		VIS.sBadPackageReason1 :=	CONCAT(CONCAT(CONCAT(CONCAT(CONCAT(CONCAT(sBadPackage1Reason1,':'),INT_TO_STRING(iBadPackage1ReasonCount1)),';'),sBadPackage2Reason1),':'),INT_TO_STRING(iBadPackage2ReasonCount1));
		VIS.sBadPackageReason2 :=	CONCAT(CONCAT(CONCAT(CONCAT(CONCAT(CONCAT(sBadPackage1Reason2,':'),INT_TO_STRING(iBadPackage1ReasonCount2)),';'),sBadPackage2Reason2),':'),INT_TO_STRING(iBadPackage2ReasonCount2));
		VIS.sBadPackageReason3 :=	CONCAT(CONCAT(CONCAT(CONCAT(CONCAT(CONCAT(sBadPackage1Reason3,':'),INT_TO_STRING(iBadPackage1ReasonCount3)),';'),sBadPackage2Reason3),':'),INT_TO_STRING(iBadPackage2ReasonCount3));
		
		
		bAddBadPackageReason	:= FALSE;
		
*)
END_ACTION

ACTION aCycleLogicHMI:
(*
Nazwa:			aCycleLogicHMI
Opis:			Wypracowanie sygnałów dla HMI
Wersja:			v0.2
Data:			2019-07-16
Autor:			DP
Urzadzenia:		
Konfiguracja:	
Info:
-daodano wbijak nasadek
*)



(*Dane do wykresów*)
//Wykresy wag i ilości wydozowanych
VIS.lrDispencer1DoseVolumeCV;			//Wartość wydana dozownika 1
VIS.lrDispencer2DoseVolumeCV;			//Wartość wydana dozownika 2
VIS.lrDispencer3DoseVolumeCV;			//Wartość wydana dozownika 3
VIS.lrDispencer4DoseVolumeCV;			//Wartość wydana dozownika 4
VIS.lrDispencer1WeightMeasured;			//Wartoć zmierzonej wagi dozowika 1 	
VIS.lrDispencer2WeightMeasured;			//Wartoć zmierzonej wagi dozowika 2	
VIS.lrDispencer3WeightMeasured;			//Wartoć zmierzonej wagi dozowika 3	
VIS.lrDispencer4WeightMeasured;			//Wartoć zmierzonej wagi dozowika 4	


//Pomiary przebiegu dozowania dozownika 1
VIS.bHMIDispencer1SuckingValveActuator					:= P02_Dispencers.QbDispencer1SuckingValveActuator;
VIS.bHMIDispencer1DosingValveActuator					:= P02_Dispencers.QbDispencer1DosingValveActuator;
VIS.bHMIDispencer1DropCatcherValveActuator				:= P02_Dispencers.QbDispencer1DropCatcherValveActuator;

//Pomiary przebiegu dozowania dozownika 2
VIS.bHMIDispencer2SuckingValveActuator					:= P02_Dispencers.QbDispencer2SuckingValveActuator;
VIS.bHMIDispencer2DosingValveActuator					:= P02_Dispencers.QbDispencer2DosingValveActuator;
VIS.bHMIDispencer2DropCatcherValveActuator				:= P02_Dispencers.QbDispencer2DropCatcherValveActuator;

//Pomiary przebiegu dozowania dozownika 3
VIS.bHMIDispencer3SuckingValveActuator					:= P02_Dispencers.QbDispencer3SuckingValveActuator;
VIS.bHMIDispencer3DosingValveActuator					:= P02_Dispencers.QbDispencer3DosingValveActuator;
VIS.bHMIDispencer3DropCatcherValveActuator				:= P02_Dispencers.QbDispencer3DropCatcherValveActuator;

//Pomiary przebiegu dozowania dozownika 3
VIS.bHMIDispencer4SuckingValveActuator					:= P02_Dispencers.QbDispencer4SuckingValveActuator;
VIS.bHMIDispencer4DosingValveActuator					:= P02_Dispencers.QbDispencer4DosingValveActuator;
VIS.bHMIDispencer4DropCatcherValveActuator				:= P02_Dispencers.QbDispencer4DropCatcherValveActuator;


(*Komunikacyjne*)
VIS.iHMICommunication:=VIS.iHMICommunication+1;

sHomingText:='';

(*Generowanie opisów przy bazowaniu*)

IF (P00_PackML.fbPMLAuto.ePMLState = E_PMLState.ePMLState_RESETTING  AND bRecipeChangePositioning AND NOT P00_PackML.iHomingCase=20) OR NOT bFirstPositioningDone   THEN
	
	IF NOT P01_BottleFeeder.fbBottleFeeder.bHomingDone OR bBottleFeederEnable THEN
		;//sHomingText:=Concat(sHomingText,'SORB,'); 
		END_IF
		
	IF NOT P01_PucksInserter.fbPucksInserter.bHomingDone OR bPucksInserterEnable THEN
		sHomingText:=Concat(sHomingText,'PI,'); END_IF
		
	IF (NOT stBottleSorterRead.bHomingDone OR stBottleSorterRead.bEnable) AND NOT bBottleSorterDisable THEN
		sHomingText:=Concat(sHomingText,'SORB,'); END_IF
		
	IF NOT P02_Dispencers.fbDispencer1.bHomingDone OR bDispencer1Enable THEN
		sHomingText:=Concat(sHomingText,'D1,'); END_IF
		
	IF NOT P02_Dispencers.fbDispencer2.bHomingDone OR bDispencer2Enable THEN
		sHomingText:=Concat(sHomingText,'D2,'); END_IF
		
	IF NOT P02_Dispencers.fbDispencer3.bHomingDone AND bDispencer3Enable THEN
		sHomingText:=Concat(sHomingText,'D3,'); END_IF
		
	IF NOT P02_Dispencers.fbDispencer4.bHomingDone AND bDispencer4Enable THEN
		sHomingText:=Concat(sHomingText,'D4,'); END_IF	
		
	IF NOT P02_Dispencers.fbDispencersDragRightStation.bHomingDone AND GVL.bFormsDragingRightEnable THEN
		sHomingText:=Concat(sHomingText,'PFDP,'); END_IF	

	IF NOT P02_Dispencers.fbDispencersDragLeftStation.bHomingDone AND GVL.bFormsDragingLeftEnable THEN
		sHomingText:=Concat(sHomingText,'PFDL,'); END_IF	
	
	IF NOT P02_Dispencers.fbDispencersCatch1Station.bHomingDone OR NOT P02_Dispencers.fbDispencersCatch2Station.bHomingDone OR NOT P02_Dispencers.fbDispencersCatch3Station.bHomingDone OR NOT P02_Dispencers.fbDispencersCatch4Station.bHomingDone OR bDispencer1Enable OR bDispencer2Enable OR bDispencer3Enable OR bDispencer4Enable THEN
		sHomingText:=Concat(sHomingText,'CHD,'); END_IF
		
	IF NOT P05_Weight.fbWeightStation.bHomingDone OR GVL.bWeightLiftEnable THEN	
		sHomingText:=Concat(sHomingText,'W,'); END_IF
	
	IF (NOT stCapSorterRead.bHomingDone OR stCapSorterRead.bEnable) AND NOT bCapSorterDisable THEN
		sHomingText:=Concat(sHomingText,'SORN,'); END_IF		

	IF	NOT P06_WickFeeder.fbWickFeederDragStation.bHomingDone AND bWickFeederDragingStationEnable THEN
		sHomingText:=Concat(sHomingText,'PPPK,'); END_IF		

	IF NOT P06_WickFeeder.fbWickFeederSt.bHomingDone AND bWickFeederEnable THEN
		sHomingText:=Concat(sHomingText,'PK,'); END_IF				

	IF NOT P06_LidFeeder.fbLidFeeder.bHomingDone AND GVL.bLidFeederEnable THEN
		sHomingText:=Concat(sHomingText,'PP1,'); END_IF			
		
	IF NOT P06_LidFeeder.fbLidFeeder2.bHomingDone AND GVL.bLidFeederEnable THEN
		sHomingText:=Concat(sHomingText,'PP2,'); END_IF			
		
	IF NOT P06_LidFeeder.fbLidFeederDragStation.bHomingDone AND GVL.bLidFeederDragingStationEnable THEN
		sHomingText:=Concat(sHomingText,'PFPP,'); END_IF			

	IF NOT P06_LidPuttedCheck.fbLidPuttedCheck.bHomingDone AND GVL.bLidPuttedCheckEnable THEN
		sHomingText:=Concat(sHomingText,'SP,'); END_IF			
		
	IF NOT P06_LidSealer.fbLidSealer.bHomingDone AND GVL.bLidSealerEnable THEN
		sHomingText:=Concat(sHomingText,'ZP1,'); END_IF			

	IF NOT P06_LidSealer.fbLidSealer2.bHomingDone AND GVL.bLidSealerEnable THEN
		sHomingText:=Concat(sHomingText,'ZP2,'); END_IF			

	IF NOT P06_LidSealer.fbLidSealerDragStation.bHomingDone AND GVL.bLidSealerDragingStationEnable THEN
		sHomingText:=Concat(sHomingText,'PFPZP,'); END_IF			

	IF NOT P07_ROPP.fbROPPFeeder.bHomingDone AND bROPPFeederEnable THEN
		sHomingText:=Concat(sHomingText,'ROPPF,'); END_IF			
	IF NOT P07_ROPP.fbROPPDrag.bHomingDone AND bROPPDragEnable THEN
		sHomingText:=Concat(sHomingText,'ROPPD,'); END_IF		
	IF NOT P07_ROPP.fbROPPCapping.bHomingDone AND bROPPCappingEnable THEN
		sHomingText:=Concat(sHomingText,'ROPPC,'); END_IF	

	IF NOT P08_CapSorter.fbCapSorterDragStation.bHomingDone AND GVL.bCapSorterDragEnable THEN
		sHomingText:=Concat(sHomingText,'PFSORN,'); END_IF	
		
	IF NOT P09_CapPuttedCheck.fbCapPuttedCheck.bHomingDone OR bCapPuttedCheckEnable THEN	
		sHomingText:=Concat(sHomingText,'SN,'); END_IF

	IF NOT P10_GripperScrewer.fbGripperScrewersDragStation.bHomingDone OR bBottleDragingStationEnable THEN	
		sHomingText:=Concat(sHomingText,'PFPZ,'); END_IF	
		
	IF NOT P10_GripperScrewer.fb2GripperScrewer1.bHomingDone OR bGripperScrewer1Enable THEN	
		sHomingText:=Concat(sHomingText,'ZS1,'); END_IF	

	IF NOT P10_GripperScrewer.fb2GripperScrewer2.bHomingDone OR bGripperScrewer2Enable THEN	
		sHomingText:=Concat(sHomingText,'ZS2,'); END_IF	
		
	IF( NOT P10_GripperScrewer.fbGripperScrewer1CatchStation.bHomingDone AND NOT P10_GripperScrewer.fbGripperScrewer2CatchStation.bHomingDone ) OR bGripperScrewer1Enable OR bGripperScrewer2Enable THEN	
		sHomingText:=Concat(sHomingText,'CHZS,'); END_IF
			
	IF NOT P11_CapCorrectCheck.fbCapCorrectCheck.bHomingDone OR bCapCorrectCheckEnable THEN	
		sHomingText:=Concat(sHomingText,'SZA,'); END_IF
		
	IF (NOT bFirstPositioningDone OR GVL.bGateRobotEnable)  THEN
		sHomingText:=Concat(sHomingText,'SZR,'); END_IF
		
	IF (NOT P13_BottleTransfer.fbBottleTransfer.bHomingDone OR bBottleTransferEnable)  THEN
		sHomingText:=Concat(sHomingText,'R,'); END_IF

ELSIF (P00_PackML.fbPMLAuto.ePMLState = E_PMLState.ePMLState_RESETTING  AND bRecipeChangePositioning) OR NOT bFirstPositioningDone OR NOT P00_PackML.bHomingIsOnAtLeastOneStation  THEN
	
	IF NOT P01_BottleFeeder.fbBottleFeeder.bHomingDone AND bBottleFeederEnable THEN
		sHomingText:=Concat(sHomingText,'SORB,'); END_IF

	IF NOT P01_PucksInserter.fbPucksInserter.bHomingDone AND bPucksInserterEnable THEN
		sHomingText:=Concat(sHomingText,'PI,'); END_IF

	IF (NOT stBottleSorterRead.bHomingDone AND stBottleSorterRead.bEnable) AND NOT bBottleSorterDisable THEN
		sHomingText:=Concat(sHomingText,'SORB,'); END_IF
		
	IF NOT P02_Dispencers.fbDispencer1.bHomingDone AND bDispencer1Enable THEN
		sHomingText:=Concat(sHomingText,'D1,'); END_IF
		
	IF NOT P02_Dispencers.fbDispencer2.bHomingDone AND bDispencer2Enable THEN
		sHomingText:=Concat(sHomingText,'D2,'); END_IF
		
	IF NOT P02_Dispencers.fbDispencer3.bHomingDone AND bDispencer3Enable THEN
		sHomingText:=Concat(sHomingText,'D3,'); END_IF
		
	IF NOT P02_Dispencers.fbDispencer4.bHomingDone AND bDispencer4Enable THEN
		sHomingText:=Concat(sHomingText,'D4,'); END_IF	
		
	IF NOT P02_Dispencers.fbDispencersDragRightStation.bHomingDone AND GVL.bFormsDragingRightEnable THEN
		sHomingText:=Concat(sHomingText,'PFDP,'); END_IF	

	IF NOT P02_Dispencers.fbDispencersDragLeftStation.bHomingDone AND GVL.bFormsDragingLeftEnable THEN
		sHomingText:=Concat(sHomingText,'PFDL,'); END_IF	
	
	IF (NOT P02_Dispencers.fbDispencersCatch1Station.bHomingDone OR NOT P02_Dispencers.fbDispencersCatch2Station.bHomingDone OR NOT P02_Dispencers.fbDispencersCatch3Station.bHomingDone OR NOT P02_Dispencers.fbDispencersCatch4Station.bHomingDone) AND (bDispencer1Enable OR bDispencer2Enable OR bDispencer3Enable OR bDispencer4Enable) THEN
		sHomingText:=Concat(sHomingText,'CHD,'); END_IF
		
	IF NOT P05_Weight.fbWeightStation.bHomingDone AND GVL.bWeightLiftEnable THEN	
		sHomingText:=Concat(sHomingText,'W,'); END_IF
	
	IF (NOT stCapSorterRead.bHomingDone AND stCapSorterRead.bEnable) AND NOT bCapSorterDisable THEN
		sHomingText:=Concat(sHomingText,'SORN,'); END_IF		


	(*IF NOT P06_LidFeeder.fbLidFeeder.bHomingDone AND GVL.bLidFeederEnable THEN
		sHomingText:=Concat(sHomingText,'PP1,'); END_IF			
		
	IF NOT P06_LidFeeder.fbLidFeeder2.bHomingDone AND GVL.bLidFeederEnable THEN
		sHomingText:=Concat(sHomingText,'PP2,'); END_IF			
		
	IF NOT P06_LidFeeder.fbLidFeederDragStation.bHomingDone AND GVL.bLidFeederDragingStationEnable THEN
		sHomingText:=Concat(sHomingText,'PFPP,'); END_IF	*)		
		
	IF	NOT P06_WickFeeder.fbWickFeederDragStation.bHomingDone AND bWickFeederDragingStationEnable THEN
		sHomingText:=Concat(sHomingText,'PPPK,'); END_IF		

	IF NOT P06_WickFeeder.fbWickFeederSt.bHomingDone AND bWickFeederEnable THEN
		sHomingText:=Concat(sHomingText,'PK,'); END_IF			
		
	IF (NOT P06_LidFeeder.fbLidFeeder.bHomingDone AND GVL.bLidFeederEnable ) OR
		(NOT P06_LidFeeder.fbLidFeeder2.bHomingDone AND GVL.bLidFeederEnable) OR
		(NOT P06_LidFeeder.fbLidFeederDragStation.bHomingDone AND GVL.bLidFeederDragingStationEnable)
	THEN
		sHomingText:=Concat(sHomingText,'PP1,'); 			
		sHomingText:=Concat(sHomingText,'PP2,'); 					
		sHomingText:=Concat(sHomingText,'PFPP,'); END_IF		
		
	IF NOT P06_LidPuttedCheck.fbLidPuttedCheck.bHomingDone AND GVL.bLidPuttedCheckEnable THEN
		sHomingText:=Concat(sHomingText,'SP,'); END_IF			
		
	IF NOT P06_LidSealer.fbLidSealer.bHomingDone AND GVL.bLidSealerEnable THEN
		sHomingText:=Concat(sHomingText,'ZP1,'); END_IF			

	IF NOT P06_LidSealer.fbLidSealer2.bHomingDone AND GVL.bLidSealerEnable THEN
		sHomingText:=Concat(sHomingText,'ZP2,'); END_IF			

	IF NOT P06_LidSealer.fbLidSealerDragStation.bHomingDone AND GVL.bLidSealerDragingStationEnable THEN
		sHomingText:=Concat(sHomingText,'PFPZP,'); END_IF			

	IF NOT P07_ROPP.fbROPPFeeder.bHomingDone AND bROPPFeederEnable THEN
		sHomingText:=Concat(sHomingText,'ROPPF,'); END_IF			
	IF NOT P07_ROPP.fbROPPDrag.bHomingDone AND bROPPDragEnable THEN
		sHomingText:=Concat(sHomingText,'ROPPD,'); END_IF		
	IF NOT P07_ROPP.fbROPPCapping.bHomingDone AND bROPPCappingEnable THEN
		sHomingText:=Concat(sHomingText,'ROPPC,'); END_IF	
	
	IF NOT P08_CapSorter.fbCapSorterDragStation.bHomingDone AND GVL.bCapSorterDragEnable THEN
		sHomingText:=Concat(sHomingText,'PFSORN,'); END_IF	
		
	IF NOT P09_CapPuttedCheck.fbCapPuttedCheck.bHomingDone AND bCapPuttedCheckEnable THEN	
		sHomingText:=Concat(sHomingText,'SN,'); END_IF

	IF NOT P10_GripperScrewer.fbGripperScrewersDragStation.bHomingDone AND bBottleDragingStationEnable THEN	
		sHomingText:=Concat(sHomingText,'PFPZ,'); END_IF	
		
	IF NOT P10_GripperScrewer.fb2GripperScrewer1.bHomingDone AND bGripperScrewer1Enable THEN	
		sHomingText:=Concat(sHomingText,'ZS1,'); END_IF	

	IF NOT P10_GripperScrewer.fb2GripperScrewer2.bHomingDone AND bGripperScrewer2Enable THEN	
		sHomingText:=Concat(sHomingText,'ZS2,'); END_IF	
		
	IF( NOT P10_GripperScrewer.fbGripperScrewer1CatchStation.bHomingDone AND NOT P10_GripperScrewer.fbGripperScrewer2CatchStation.bHomingDone ) AND (bGripperScrewer1Enable OR bGripperScrewer2Enable) THEN	
		sHomingText:=Concat(sHomingText,'CHZS,'); END_IF
			
	IF NOT P11_CapCorrectCheck.fbCapCorrectCheck.bHomingDone AND bCapCorrectCheckEnable THEN	
		sHomingText:=Concat(sHomingText,'SZA,'); END_IF
		
	IF (NOT bFirstPositioningDone AND GVL.bGateRobotEnable)  THEN
		sHomingText:=Concat(sHomingText,'SZR,'); END_IF
		
	IF (NOT P13_BottleTransfer.fbBottleTransfer.bHomingDone AND bBottleTransferEnable)  THEN
		sHomingText:=Concat(sHomingText,'R,'); END_IF
		
ELSIF P00_PackML.fbPMLAuto.ePMLState = E_PMLState.ePMLState_RESETTING AND NOT bRecipeChangePositioning AND P00_Visualization.iCaseDialogHoming = 10 THEN
	
	IF stBottleSorterWrite.bHoming AND stBottleSorterRead.bEnable AND NOT bBottleSorterDisable THEN
		sHomingText:=Concat(sHomingText,'SORB,'); END_IF

	IF VIS.bPucksInserterHoming AND bPucksInserterEnable THEN
		sHomingText:=Concat(sHomingText,'PI,'); END_IF

	IF VIS.bDispencersHoming AND bDispencer1Enable THEN
		sHomingText:=Concat(sHomingText,'D1,'); END_IF
		
	IF VIS.bDispencersHoming AND bDispencer2Enable THEN
		sHomingText:=Concat(sHomingText,'D2,'); END_IF
		
	IF VIS.bDispencersHoming AND bDispencer3Enable THEN
		sHomingText:=Concat(sHomingText,'D3,'); END_IF
		
	IF VIS.bDispencersHoming AND bDispencer4Enable THEN
		sHomingText:=Concat(sHomingText,'D4,'); END_IF
		
	IF VIS.bFormsDragingRightHoming AND GVL.bFormsDragingRightEnable THEN
		sHomingText:=Concat(sHomingText,'PFDP,'); END_IF

	IF VIS.bFormsDragingLeftHoming AND GVL.bFormsDragingLeftEnable THEN
		sHomingText:=Concat(sHomingText,'PFDL,'); END_IF
			
	IF VIS.bDispencersHoming THEN
		sHomingText:=Concat(sHomingText,'CHD,'); END_IF
		
	IF VIS.bWeightLiftHoming THEN	
		sHomingText:=Concat(sHomingText,'W,'); END_IF	
		
	IF VIS.bWickFeederHoming THEN
		sHomingText:=Concat(sHomingText,'PK,'); END_IF			
		
	IF VIS.bWickFeederDragingHoming  THEN
		sHomingText:=Concat(sHomingText,'PPPK,'); END_IF			

	IF VIS.bLidFeederHoming OR VIS.bLidFeederDragingHoming THEN
		sHomingText:=Concat(sHomingText,'PP1,PP2,'); END_IF			
		
	IF VIS.bLidFeederDragingHoming OR VIS.bLidFeederHoming THEN
		sHomingText:=Concat(sHomingText,'PFPP,'); END_IF			

	IF VIS.bLidPuttedCheckHoming THEN
		sHomingText:=Concat(sHomingText,'SP,'); END_IF			
		
	IF VIS.bLidSealerHoming THEN
		sHomingText:=Concat(sHomingText,'ZP1,ZP2,'); END_IF			

	IF VIS.bLidSealerDragingHoming THEN
		sHomingText:=Concat(sHomingText,'PFPZP,'); END_IF					
	
	IF VIS_ROPP.bROPPFeederHoming  AND bROPPFeederEnable THEN
		sHomingText:=Concat(sHomingText,'ROPPF,'); END_IF			
	IF VIS_ROPP.bROPPDragHoming AND bROPPDragEnable THEN
		sHomingText:=Concat(sHomingText,'ROPPD,'); END_IF		
	IF VIS_ROPP.bROPPCappingHoming AND bROPPCappingEnable THEN
		sHomingText:=Concat(sHomingText,'ROPPC,'); END_IF	

	IF stCapSorterWrite.bHoming AND stCapSorterRead.bEnable AND NOT bCapSorterDisable THEN
		sHomingText:=Concat(sHomingText,'SORN,'); END_IF		
		
	IF VIS.bCapSorterDragHoming AND GVL.bCapSorterDragEnable THEN
		sHomingText:=Concat(sHomingText,'PFSORN,'); END_IF	
		
	IF VIS.bCapPuttedCheckHoming THEN	
		sHomingText:=Concat(sHomingText,'CC,'); END_IF

	IF VIS.bBottleDragingStationHoming AND GVL.bBottleDragingStationEnable THEN
		sHomingText:=Concat(sHomingText,'PFPZ,'); END_IF
		
	IF VIS.bGripperScrewerHoming THEN	
		sHomingText:=Concat(sHomingText,'ZS,'); END_IF	
		
	IF VIS.bGripperScrewerHoming THEN	
		sHomingText:=Concat(sHomingText,'CHZS,'); END_IF
		
	IF VIS.bCapCorrectCheckHoming THEN	
		sHomingText:=Concat(sHomingText,'SZA,'); END_IF
		
	IF (VIS.bBottleTransferHoming)  THEN
		sHomingText:=Concat(sHomingText,'R,'); END_IF
		
	IF (VIS.bCapFeederHoming) THEN
		sHomingText:=Concat(sHomingText,'PN,'); END_IF

	
ELSE
	sHomingText:='';
END_IF




(*Rejestry**********************************************************************)
VIS.AbFormPresent[1]			:=	eBottleFeederPackageState[1].bFormPresent;
VIS.AsFormDescription[1]		:=	FormDescription	(
														B:=	eBottleFeederPackageState[1].bBottlePresent,
														W:=	0,	
														N:=	0, 
														Z:=	0
													);
									
(*****Nastepny**************************************************************************)									
VIS.AbFormPresent[2]			:=	(eBeforeDispencersPackageState[4].bFormPresent AND NOT bDosingTwoPhases)  OR (eBeforeDispencer34PackageState2Phase[2].bFormPresent AND bDosingTwoPhases);
 VIS.AsFormDescription[2]		:=	FormDescription	(
														B:=(eBeforeDispencersPackageState[4].bBottlePresent AND NOT bDosingTwoPhases) OR (eBeforeDispencer34PackageState2Phase[2].bBottlePresent AND bDosingTwoPhases), 
														W:=	0,	
														N:=	0, 
														Z:=	0
													);																																	
VIS.AbFormPresent[3]			:=	(eBeforeDispencersPackageState[3].bFormPresent AND NOT bDosingTwoPhases)  OR (eBeforeDispencer34PackageState2Phase[1].bFormPresent AND bDosingTwoPhases);
VIS.AsFormDescription[3]		:=	FormDescription	(
														B:=(eBeforeDispencersPackageState[3].bBottlePresent AND NOT bDosingTwoPhases) OR (eBeforeDispencer34PackageState2Phase[1].bBottlePresent AND bDosingTwoPhases),
														W:=	0,	
														N:=	0, 
														Z:=	0
													);																						
VIS.AbFormPresent[4]			:=	(eBeforeDispencersPackageState[2].bFormPresent AND NOT bDosingTwoPhases)  OR (eAfterDispencer12PackageState2Phase[2].bFormPresent AND bDosingTwoPhases);
VIS.AsFormDescription[4]		:=	FormDescription	(
														B:=(eBeforeDispencersPackageState[2].bBottlePresent AND NOT bDosingTwoPhases) OR (eAfterDispencer12PackageState2Phase[1].bBottlePresent AND bDosingTwoPhases),
														W:=	0,	
														N:=	0, 
														Z:=	0
													);																					
VIS.AbFormPresent[5]			:=	(eBeforeDispencersPackageState[1].bFormPresent AND NOT bDosingTwoPhases)  OR (eAfterDispencer12PackageState2Phase[1].bFormPresent AND bDosingTwoPhases) ;
VIS.AsFormDescription[5]		:=	FormDescription	(
														B:=(eBeforeDispencersPackageState[1].bBottlePresent AND NOT bDosingTwoPhases) OR (eAfterDispencer12PackageState2Phase[2].bBottlePresent AND bDosingTwoPhases),
														W:=	0,	
														N:=	0, 
														Z:=	0
													);									
(*****Nastepny**************************************************************************)															
                                                              	
VIS.AbFormPresent[6]			:=	(eDispencersPackageState[4].bFormPresent AND NOT bDosingTwoPhases) OR (eDispencer34PackageState2Phase[2].bFormPresent AND bDosingTwoPhases);
VIS.AsFormDescription[6]		:=	FormDescription	(
														B:=(eDispencersPackageState[4].bBottlePresent AND NOT bDosingTwoPhases) OR (eDispencer34PackageState2Phase[2].bBottlePresent AND bDosingTwoPhases),
														W:=	0,	
														N:=	0, 
														Z:=	0
													);			

VIS.AbFormPresent[7]			:=	(eDispencersPackageState[3].bFormPresent AND NOT bDosingTwoPhases) OR (eDispencer34PackageState2Phase[1].bFormPresent AND bDosingTwoPhases);
VIS.AsFormDescription[7]		:=	FormDescription	(
														B:=(eDispencersPackageState[3].bBottlePresent AND NOT bDosingTwoPhases) OR (eDispencer34PackageState2Phase[1].bBottlePresent AND bDosingTwoPhases),
														W:=	0,	
														N:=	0, 
														Z:=	0
													);			

VIS.AbFormPresent[8]			:=	(eDispencersPackageState[2].bFormPresent AND NOT bDosingTwoPhases) OR (eDispencer12PackageState2Phase[2].bFormPresent AND bDosingTwoPhases);
VIS.AsFormDescription[8]		:=	FormDescription	(
														B:=(eDispencersPackageState[2].bBottlePresent AND NOT bDosingTwoPhases) OR (eDispencer12PackageState2Phase[2].bBottlePresent AND bDosingTwoPhases),
														W:=	0,	
														N:=	0, 
														Z:=	0
													);			

VIS.AbFormPresent[9]			:=	(eDispencersPackageState[1].bFormPresent AND NOT bDosingTwoPhases) OR (eDispencer12PackageState2Phase[1].bFormPresent AND bDosingTwoPhases);
VIS.AsFormDescription[9]		:=	FormDescription	(
														B:=(eDispencersPackageState[1].bBottlePresent AND NOT bDosingTwoPhases) OR (eDispencer12PackageState2Phase[1].bBottlePresent AND bDosingTwoPhases),
														W:=	0,	
														N:=	0, 
														Z:=	0
													);			
  (*****Nastepny**************************************************************************)                                                            	
VIS.AbFormPresent[10]  			:=	(eAfterDispencersPackageState[4].bFormPresent AND NOT bDosingTwoPhases)  OR (eAfterDispencer34PackageState2Phase[2].bFormPresent AND bDosingTwoPhases);
VIS.AsFormDescription[10]		:=	FormDescription	(
														B:=	(eAfterDispencersPackageState[4].bBottlePresent AND NOT bDosingTwoPhases)	OR (eAfterDispencer34PackageState2Phase[2].bBottlePresent AND bDosingTwoPhases),
														W:=	0,	
														N:=	0, 
														Z:=	0
													);		
VIS.AbFormPresent[11] 			:=	(eAfterDispencersPackageState[3].bFormPresent AND NOT bDosingTwoPhases)  OR (eAfterDispencer34PackageState2Phase[1].bFormPresent AND bDosingTwoPhases);
VIS.AsFormDescription[11]		:=	FormDescription	(
														B:=	(eAfterDispencersPackageState[3].bBottlePresent AND NOT bDosingTwoPhases)	OR (eAfterDispencer34PackageState2Phase[1].bBottlePresent AND bDosingTwoPhases),
														W:=	0,	
														N:=	0, 
														Z:=	0
													);		
VIS.AbFormPresent[12] 			:=	(eAfterDispencersPackageState[2].bFormPresent AND NOT bDosingTwoPhases)  OR (eBeforeDispencer12PackageState2Phase[2].bFormPresent AND bDosingTwoPhases);
VIS.AsFormDescription[12]		:=	FormDescription	(
														B:=	(eAfterDispencersPackageState[2].bBottlePresent AND NOT bDosingTwoPhases)	OR (eBeforeDispencer12PackageState2Phase[2].bBottlePresent AND bDosingTwoPhases),
														W:=	0,	
														N:=	0, 
														Z:=	0
													);		
VIS.AbFormPresent[13]  			:=	(eAfterDispencersPackageState[1].bFormPresent AND NOT bDosingTwoPhases)  OR (eBeforeDispencer12PackageState2Phase[1].bFormPresent AND bDosingTwoPhases);
VIS.AsFormDescription[13]		:=	FormDescription	(
														B:=	(eAfterDispencersPackageState[1].bBottlePresent AND NOT bDosingTwoPhases)	OR (eBeforeDispencer12PackageState2Phase[1].bBottlePresent AND bDosingTwoPhases),
														W:=	0,	
														N:=	0, 
														Z:=	0
													);		
(*****Nastepny**************************************************************************)                                                             	
VIS.AbFormPresent[14]			:=	eWeightPackageState[4].bFormPresent;
VIS.AsFormDescription[14]		:=	FormDescription	(
														B:=	eWeightPackageState[4].bBottlePresent,
														W:=	eWeightPackageState[4].bWeightOK,	
														N:=	0, 
														Z:=	0
													);		
VIS.AbFormPresent[15] 			:=	eWeightPackageState[3].bFormPresent;
VIS.AsFormDescription[15]		:=	FormDescription	(
														B:=	eWeightPackageState[3].bBottlePresent,
														W:=	eWeightPackageState[3].bWeightOK,	
														N:=	0, 
														Z:=	0
													);		
VIS.AbFormPresent[16] 			:=	eWeightPackageState[2].bFormPresent;
VIS.AsFormDescription[16]		:=	FormDescription	(
														B:=	eWeightPackageState[2].bBottlePresent,
														W:=	eWeightPackageState[2].bWeightOK,	
														N:=	0, 
														Z:=	0
													);		
VIS.AbFormPresent[17]  			:=	eWeightPackageState[1].bFormPresent;
VIS.AsFormDescription[17]		:=	FormDescription	(
														B:=	eWeightPackageState[1].bBottlePresent,
														W:=	eWeightPackageState[1].bWeightOK,	
														N:=	0, 
														Z:=	0
													);	
(*****Nastepny**************************************************************************)
VIS.AbFormPresent[18]			:=	eWeightPackage2PhasePackageState[2].bFormPresent;
VIS.AsFormDescription[18]		:=	FormDescription	(
														B:=	eWeightPackage2PhasePackageState[2].bBottlePresent,
														W:=	eWeightPackage2PhasePackageState[2].bWeightOK,	
														N:=	0, 
														Z:=	0
													);		
VIS.AbFormPresent[19]			:=	eWeightPackage2PhasePackageState[1].bFormPresent;
VIS.AsFormDescription[19]		:=	FormDescription	(
														B:=	eWeightPackage2PhasePackageState[1].bBottlePresent,
														W:=	eWeightPackage2PhasePackageState[1].bWeightOK,	
														N:=	0, 
														Z:=	0
													);		
													
(*****Nastepny**************************************************************************)                                                             	
VIS.AbFormPresent[20] 			:=	eBeforeGateCapSorterPackageState[1].bFormPresent;
VIS.AsFormDescription[20]		:=	FormDescription	(
														B:=	eBeforeGateCapSorterPackageState[1].bBottlePresent,
														W:=	eBeforeGateCapSorterPackageState[1].bWeightOK,	
														N:=	0,
														Z:=	0
													);						
(*****Nastepny**************************************************************************)     									
VIS.AbFormPresent[21] 			:=	eBeforeCapSorterPackageState[4].bFormPresent;
VIS.AsFormDescription[21]		:=	FormDescription	(
														B:=	eBeforeCapSorterPackageState[4].bBottlePresent,
														W:=	eBeforeCapSorterPackageState[4].bWeightOK,	
														N:=	0,
														Z:=	0
													);															
VIS.AbFormPresent[22] 			:=	eBeforeCapSorterPackageState[3].bFormPresent;
VIS.AsFormDescription[22]		:=	FormDescription	(
														B:=	eBeforeCapSorterPackageState[3].bBottlePresent,
														W:=	eBeforeCapSorterPackageState[3].bWeightOK,	
														N:=	0,
														Z:=	0
													);																	
VIS.AbFormPresent[23] 			:=	eBeforeCapSorterPackageState[2].bFormPresent;
VIS.AsFormDescription[23]		:=	FormDescription	(
														B:=	eBeforeCapSorterPackageState[2].bBottlePresent,
														W:=	eBeforeCapSorterPackageState[2].bWeightOK,	
														N:=	0,
														Z:=	0
													);															
VIS.AbFormPresent[24] 			:=	eBeforeCapSorterPackageState[1].bFormPresent;
VIS.AsFormDescription[24]		:=	FormDescription	(
														B:=	eBeforeCapSorterPackageState[1].bBottlePresent,
														W:=	eBeforeCapSorterPackageState[1].bWeightOK,	
														N:=	0,
														Z:=	0
													);																																																					
(*****Nastepny**************************************************************************)     									
VIS.AbFormPresent[25] 			:=	eCapSorterPackageState[4].bFormPresent;
VIS.AsFormDescription[25]		:=	FormDescription	(
														B:=	eCapSorterPackageState[4].bBottlePresent,
														W:=	eCapSorterPackageState[4].bWeightOK,	
														N:=	eCapSorterPackageState[4].bCapSorterPutted,
														Z:=	0
													);															
VIS.AbFormPresent[26] 			:=	eCapSorterPackageState[3].bFormPresent;
VIS.AsFormDescription[26]		:=	FormDescription	(
														B:=	eCapSorterPackageState[3].bBottlePresent,
														W:=	eCapSorterPackageState[3].bWeightOK,	
														N:=	eCapSorterPackageState[3].bCapSorterPutted,
														Z:=	0
													);																	
VIS.AbFormPresent[27] 			:=	eCapSorterPackageState[2].bFormPresent;
VIS.AsFormDescription[27]		:=	FormDescription	(
														B:=	eCapSorterPackageState[2].bBottlePresent,
														W:=	eCapSorterPackageState[2].bWeightOK,	
														N:=	eCapSorterPackageState[2].bCapSorterPutted,
														Z:=	0
													);															
VIS.AbFormPresent[28] 			:=	eCapSorterPackageState[1].bFormPresent;
VIS.AsFormDescription[28]		:=	FormDescription	(
														B:=	eCapSorterPackageState[1].bBottlePresent,
														W:=	eCapSorterPackageState[1].bWeightOK,	
														N:=	eCapSorterPackageState[1].bCapSorterPutted,
														Z:=	0
													);					
(*****Nastepny**************************************************************************)     									
VIS.AbFormPresent[29] 			:=	eAfterCapSorterPackageState[4].bFormPresent;
VIS.AsFormDescription[29]		:=	FormDescription	(
														B:=	eAfterCapSorterPackageState[4].bBottlePresent,
														W:=	eAfterCapSorterPackageState[4].bWeightOK,	
														N:=	eAfterCapSorterPackageState[4].bCapSorterPutted,
														Z:=	0
													);															
VIS.AbFormPresent[30] 			:=	eAfterCapSorterPackageState[3].bFormPresent;
VIS.AsFormDescription[30]		:=	FormDescription	(
														B:=	eAfterCapSorterPackageState[3].bBottlePresent,
														W:=	eAfterCapSorterPackageState[3].bWeightOK,	
														N:=	eAfterCapSorterPackageState[3].bCapSorterPutted,
														Z:=	0
													);																	
VIS.AbFormPresent[31] 			:=	eAfterCapSorterPackageState[2].bFormPresent;
VIS.AsFormDescription[31]		:=	FormDescription	(
														B:=	eAfterCapSorterPackageState[2].bBottlePresent,
														W:=	eAfterCapSorterPackageState[2].bWeightOK,	
														N:=	eAfterCapSorterPackageState[2].bCapSorterPutted,
														Z:=	0
													);															
VIS.AbFormPresent[32] 			:=	eAfterCapSorterPackageState[1].bFormPresent;
VIS.AsFormDescription[32]		:=	FormDescription	(
														B:=	eAfterCapSorterPackageState[1].bBottlePresent,
														W:=	eAfterCapSorterPackageState[1].bWeightOK,	
														N:=	eAfterCapSorterPackageState[1].bCapSorterPutted,
														Z:=	0
													);		

VIS.AbFormPresent[33] 	;	
VIS.AsFormDescription[33];
VIS.AbFormPresent[34] 	;	
VIS.AsFormDescription[34];
VIS.AbFormPresent[35] 	;	
VIS.AsFormDescription[35];
				
(*****Nastepny**************************************************************************)                                                             	
VIS.AbFormPresent[36] 			:=	eBeforeScrewers2PackageState[2].bFormPresent;
VIS.AsFormDescription[36]		:=	FormDescription	(
														B:=	eBeforeScrewers2PackageState[2].bBottlePresent,
														W:=	eBeforeScrewers2PackageState[2].bWeightOK,	
														N:=	eBeforeScrewers2PackageState[2].bCapOK, 
														Z:=	0
													);		
VIS.AbFormPresent[37]			:=	eBeforeScrewers2PackageState[1].bFormPresent;
VIS.AsFormDescription[37]		:=	FormDescription	(
														B:=	eBeforeScrewers2PackageState[1].bBottlePresent,
														W:=	eBeforeScrewers2PackageState[1].bWeightOK,	
														N:=	eBeforeScrewers2PackageState[1].bCapOK, 
														Z:=	0
													);		
(*****Nastepny**************************************************************************)
VIS.AbFormPresent[38]			:=	eBeforeScrewersPackageState[2].bFormPresent;
VIS.AsFormDescription[38]		:=	FormDescription	(
														B:=	eBeforeScrewersPackageState[2].bBottlePresent,
														W:=	eBeforeScrewersPackageState[2].bWeightOK,	
														N:=	eBeforeScrewersPackageState[2].bCapOK, 
														Z:=	0
													);		
VIS.AbFormPresent[39] 			:=	eBeforeScrewersPackageState[1].bFormPresent;
VIS.AsFormDescription[39]		:=	FormDescription	(
														B:=	eBeforeScrewersPackageState[1].bBottlePresent,
														W:=	eBeforeScrewersPackageState[1].bWeightOK,	
														N:=	eBeforeScrewersPackageState[1].bCapOK, 
														Z:=	0
													);		
(*****Nastepny**************************************************************************)                                                              	
VIS.AbFormPresent[40]			:=	eUnderScrewerPackageState[2].bFormPresent;
VIS.AsFormDescription[40]		:=	FormDescription	(
														B:=	eUnderScrewerPackageState[2].bBottlePresent,
														W:=	eUnderScrewerPackageState[2].bWeightOK,	
														N:=	eUnderScrewerPackageState[2].bCapOK, 
														Z:=	eUnderScrewerPackageState[2].bCapGripperScrewed
													);		
VIS.AbFormPresent[41]  			:=	eUnderScrewerPackageState[1].bFormPresent;
VIS.AsFormDescription[41]		:=	FormDescription	(
														B:=	eUnderScrewerPackageState[1].bBottlePresent,
														W:=	eUnderScrewerPackageState[1].bWeightOK,	
														N:=	eUnderScrewerPackageState[1].bCapOK, 
														Z:=	eUnderScrewerPackageState[1].bCapGripperScrewed
													);		
(*****Nastepny**************************************************************************)                                             				  	
VIS.AbFormPresent[42]  			:=	eAfterScrewerPackageState[2].bFormPresent;
VIS.AsFormDescription[42]		:=	FormDescription	(
														B:=	eAfterScrewerPackageState[2].bBottlePresent,
														W:=	eAfterScrewerPackageState[2].bWeightOK,	
														N:=	eAfterScrewerPackageState[2].bCapCorrectCapOn AND eAfterScrewerPackageState[2].bCapOK, 
														Z:=	eAfterScrewerPackageState[2].bCapGripperScrewed
													);		
VIS.AbFormPresent[43] 			:=	eAfterScrewerPackageState[1].bFormPresent;
VIS.AsFormDescription[43]		:=	FormDescription	(
														B:=	eAfterScrewerPackageState[1].bBottlePresent,
														W:=	eAfterScrewerPackageState[1].bWeightOK,	
														N:=	eAfterScrewerPackageState[1].bCapCorrectCapOn AND eAfterScrewerPackageState[1].bCapOK, 
														Z:=	eAfterScrewerPackageState[1].bCapGripperScrewed
													);		
(*****Nastepny**************************************************************************)
VIS.AbFormPresent[44]			:=	eUnderCorrectCapPackageState[1].bFormPresent;
VIS.AsFormDescription[44]		:=	FormDescription	(
														B:= eUnderCorrectCapPackageState[1].bBottlePresent,
														W:=	eUnderCorrectCapPackageState[1].bWeightOK,	
														N:=	eUnderCorrectCapPackageState[1].bCapCorrectCapOn AND NOT eUnderCorrectCapPackageState[1].bCapCorrectNOK, 
														Z:=	eUnderCorrectCapPackageState[1].bCapGripperScrewed
													);		
VIS.AbFormPresent[45]			:=	eUnderCorrectCapPackageState[7].bFormPresent;
VIS.AsFormDescription[45]		:=	FormDescription	(
														B:=	eUnderCorrectCapPackageState[7].bBottlePresent,
														W:=	eUnderCorrectCapPackageState[7].bWeightOK,	
														N:=	eUnderCorrectCapPackageState[7].bCapCorrectCapOn AND NOT eUnderCorrectCapPackageState[7].bCapCorrectNOK, 
														Z:=	eUnderCorrectCapPackageState[7].bCapGripperScrewed
													);		
VIS.AbFormPresent[46]			:=	eUnderCorrectCapPackageState[6].bFormPresent;
VIS.AsFormDescription[46]		:=	FormDescription	(
														B:=	eUnderCorrectCapPackageState[6].bBottlePresent,
														W:=	eUnderCorrectCapPackageState[6].bWeightOK,	
														N:=	eUnderCorrectCapPackageState[6].bCapCorrectCapOn AND NOT eUnderCorrectCapPackageState[6].bCapCorrectNOK, 
														Z:=	eUnderCorrectCapPackageState[6].bCapGripperScrewed
													);		
VIS.AbFormPresent[47]			:=	eUnderCorrectCapPackageState[5].bFormPresent;
VIS.AsFormDescription[47]		:=	FormDescription	(
														B:=	eUnderCorrectCapPackageState[5].bBottlePresent,
														W:=	eUnderCorrectCapPackageState[5].bWeightOK,
														N:=	eUnderCorrectCapPackageState[5].bCapCorrectCapOn AND NOT eUnderCorrectCapPackageState[5].bCapCorrectNOK, 
														Z:=	eUnderCorrectCapPackageState[5].bCapGripperScrewed
													);		
VIS.AbFormPresent[48]			:=	eUnderCorrectCapPackageState[4].bFormPresent;
VIS.AsFormDescription[48]		:=	FormDescription	(
														B:=	eUnderCorrectCapPackageState[4].bBottlePresent,
														W:=	eUnderCorrectCapPackageState[4].bWeightOK,	
														N:=	eUnderCorrectCapPackageState[4].bCapCorrectCapOn AND NOT eUnderCorrectCapPackageState[4].bCapCorrectNOK, 
														Z:=	eUnderCorrectCapPackageState[4].bCapGripperScrewed
													);		
VIS.AbFormPresent[49]			:=	eUnderCorrectCapPackageState[3].bFormPresent;
VIS.AsFormDescription[49]		:=	FormDescription	(
														B:=	eUnderCorrectCapPackageState[3].bBottlePresent,
														W:=	eUnderCorrectCapPackageState[3].bWeightOK,	
														N:=	eUnderCorrectCapPackageState[3].bCapCorrectCapOn AND NOT eUnderCorrectCapPackageState[3].bCapCorrectNOK, 
														Z:=	eUnderCorrectCapPackageState[3].bCapGripperScrewed
													);		
VIS.AbFormPresent[50]			:=	eUnderCorrectCapPackageState[2].bFormPresent;
VIS.AsFormDescription[50]		:=	FormDescription	(
														B:=	eUnderCorrectCapPackageState[2].bBottlePresent,
														W:=	eUnderCorrectCapPackageState[2].bWeightOK,	
														N:=	eUnderCorrectCapPackageState[2].bCapCorrectCapOn AND NOT eUnderCorrectCapPackageState[2].bCapCorrectNOK, 
														Z:=	eUnderCorrectCapPackageState[2].bCapGripperScrewed
													);		
VIS.AbFormPresent[51]			:=	eUnderCorrectCapPackageState[1].bFormPresent;
VIS.AsFormDescription[51]		:=	FormDescription	(
														B:=	eUnderCorrectCapPackageState[1].bBottlePresent,
														W:=	eUnderCorrectCapPackageState[1].bWeightOK,	
														N:=	eUnderCorrectCapPackageState[1].bCapCorrectCapOn AND NOT eUnderCorrectCapPackageState[1].bCapCorrectNOK, 
														Z:=	eUnderCorrectCapPackageState[1].bCapGripperScrewed
													);									
													
 (*****Nastepny**************************************************************************)                                                             	
VIS.AbFormPresent[52]			:=	eRobotPackageState[2].bFormPresent;
VIS.AsFormDescription[52]		:=	FormDescription	(
														B:=	eRobotPackageState[2].bBottlePresent,
														W:=	eRobotPackageState[2].bWeightOK,	
														N:=	eRobotPackageState[2].bCapCorrectCapOn AND NOT eRobotPackageState[2].bCapCorrectNOK, 
														Z:=	eRobotPackageState[2].bCapGripperScrewed
													);		
VIS.AbFormPresent[53]			:=	eRobotPackageState[1].bFormPresent;
VIS.AsFormDescription[53]		:=	FormDescription	(
														B:=	eRobotPackageState[1].bBottlePresent,
														W:=	eRobotPackageState[1].bWeightOK,	
														N:=	eRobotPackageState[1].bCapCorrectCapOn AND NOT eRobotPackageState[1].bCapCorrectNOK, 
														Z:=	eRobotPackageState[1].bCapGripperScrewed
													);		
													
 (*****Nastepny**************************************************************************)                                                             	
VIS.AbFormPresent[52]			:=	eHistoryPackageState[1].bFormPresent;
VIS.AsFormDescription[52]		:=	FormDescription	(
														B:=	eHistoryPackageState[1].bBottlePresent,
														W:=	eHistoryPackageState[1].bWeightOK,	
														N:=	eHistoryPackageState[1].bCapCorrectCapOn AND NOT eRobotPackageState[2].bCapCorrectNOK, 
														Z:=	eHistoryPackageState[1].bCapGripperScrewed
													);		
VIS.AbFormPresent[53]			:=	eHistoryPackageState[2].bFormPresent;
VIS.AsFormDescription[53]		:=	FormDescription	(
														B:=	eHistoryPackageState[2].bBottlePresent,
														W:=	eHistoryPackageState[2].bWeightOK,	
														N:=	eHistoryPackageState[2].bCapCorrectCapOn AND NOT eRobotPackageState[2].bCapCorrectNOK, 
														Z:=	eHistoryPackageState[2].bCapGripperScrewed
													);
END_ACTION

ACTION aCycleLogicHMI_v2:
(*
Nazwa:			aCycleLogicHMI
Opis:			Wypracowanie sygnałów dla HMI
Wersja:			v0.2
Data:			2019-07-16
Autor:			DP
Urzadzenia:		
Konfiguracja:	
Info:
-daodano wbijak nasadek
*)
(*

(*Dane do wykresów*)
//Wykresy wag i ilości wydozowanych
VIS.lrDispencer1DoseVolumeCV;			//Wartość wydana dozownika 1
VIS.lrDispencer2DoseVolumeCV;			//Wartość wydana dozownika 2
VIS.lrDispencer3DoseVolumeCV;			//Wartość wydana dozownika 3
VIS.lrDispencer4DoseVolumeCV;			//Wartość wydana dozownika 4
VIS.lrDispencer1WeightMeasured;			//Wartoć zmierzonej wagi dozowika 1 	
VIS.lrDispencer2WeightMeasured;			//Wartoć zmierzonej wagi dozowika 2	
VIS.lrDispencer3WeightMeasured;			//Wartoć zmierzonej wagi dozowika 3	
VIS.lrDispencer4WeightMeasured;			//Wartoć zmierzonej wagi dozowika 4	


//Pomiary przebiegu dozowania dozownika 1
VIS.bHMIDispencer1SuckingValveActuator					:= P02_Dispencers.QbDispencer1SuckingValveActuator;
VIS.bHMIDispencer1DosingValveActuator					:= P02_Dispencers.QbDispencer1DosingValveActuator;
VIS.bHMIDispencer1DropCatcherValveActuator				:= P02_Dispencers.QbDispencer1DropCatcherValveActuator;

//Pomiary przebiegu dozowania dozownika 2
VIS.bHMIDispencer2SuckingValveActuator					:= P02_Dispencers.QbDispencer2SuckingValveActuator;
VIS.bHMIDispencer2DosingValveActuator					:= P02_Dispencers.QbDispencer2DosingValveActuator;
VIS.bHMIDispencer2DropCatcherValveActuator				:= P02_Dispencers.QbDispencer2DropCatcherValveActuator;

//Pomiary przebiegu dozowania dozownika 3
VIS.bHMIDispencer3SuckingValveActuator					:= P02_Dispencers.QbDispencer3SuckingValveActuator;
VIS.bHMIDispencer3DosingValveActuator					:= P02_Dispencers.QbDispencer3DosingValveActuator;
VIS.bHMIDispencer3DropCatcherValveActuator				:= P02_Dispencers.QbDispencer3DropCatcherValveActuator;

//Pomiary przebiegu dozowania dozownika 3
VIS.bHMIDispencer4SuckingValveActuator					:= P02_Dispencers.QbDispencer4SuckingValveActuator;
VIS.bHMIDispencer4DosingValveActuator					:= P02_Dispencers.QbDispencer4DosingValveActuator;
VIS.bHMIDispencer4DropCatcherValveActuator				:= P02_Dispencers.QbDispencer4DropCatcherValveActuator;


(*Komunikacyjne*)
VIS.iHMICommunication:=VIS.iHMICommunication+1;

sHomingText:='';

(*Generowanie opisów przy bazowaniu*)
IF (P00_PackML.fbPMLAuto.ePMLState = E_PMLState.ePMLState_RESETTING  AND bRecipeChangePositioning) OR NOT bFirstPositioningDone  THEN
	
	IF NOT P01_BottleFeeder.fbBottleFeeder.bHomingDone OR bBottleFeederEnable THEN
		sHomingText:=Concat(sHomingText,'SORB,'); END_IF

	IF NOT P02_Dispencers.fbDispencer1.bHomingDone OR bDispencer1Enable THEN
		sHomingText:=Concat(sHomingText,'D1,'); END_IF
		
	IF NOT P02_Dispencers.fbDispencer2.bHomingDone OR bDispencer2Enable THEN
		sHomingText:=Concat(sHomingText,'D2,'); END_IF
		
	IF NOT P02_Dispencers.fbDispencer3.bHomingDone AND bDispencer3Enable THEN
		sHomingText:=Concat(sHomingText,'D3,'); END_IF
		
	IF NOT P02_Dispencers.fbDispencer4.bHomingDone AND bDispencer4Enable THEN
		sHomingText:=Concat(sHomingText,'D4,'); END_IF	
		
	IF NOT P02_Dispencers.fbDispencersDragRightStation.bHomingDone AND GVL.bFormsDragingRightEnable THEN
		sHomingText:=Concat(sHomingText,'PFDP,'); END_IF	

	IF NOT P02_Dispencers.fbDispencersDragLeftStation.bHomingDone AND GVL.bFormsDragingLeftEnable THEN
		sHomingText:=Concat(sHomingText,'PFDL,'); END_IF	
	
	IF NOT P02_Dispencers.fbDispencersCatch1Station.bHomingDone OR NOT P02_Dispencers.fbDispencersCatch2Station.bHomingDone OR NOT P02_Dispencers.fbDispencersCatch3Station.bHomingDone OR NOT P02_Dispencers.fbDispencersCatch4Station.bHomingDone OR bDispencer1Enable OR bDispencer2Enable OR bDispencer3Enable OR bDispencer4Enable THEN
		sHomingText:=Concat(sHomingText,'CHD,'); END_IF
		
	IF NOT P05_Weight.fbWeightStation.bHomingDone OR GVL.bWeightLiftEnable THEN	
		sHomingText:=Concat(sHomingText,'W,'); END_IF
	
	IF NOT P09_CapPuttedCheck.fbCapPuttedCheck.bHomingDone OR bCapPuttedCheckEnable THEN	
		sHomingText:=Concat(sHomingText,'SN,'); END_IF

	IF NOT P10_GripperScrewer.fbGripperScrewersDragStation.bHomingDone OR bBottleDragingStationEnable THEN	
		sHomingText:=Concat(sHomingText,'PFPZ,'); END_IF	
		
	IF NOT P10_GripperScrewer.fb2GripperScrewer1.bHomingDone OR bGripperScrewer1Enable THEN	
		sHomingText:=Concat(sHomingText,'ZS1,'); END_IF	

	IF NOT P10_GripperScrewer.fb2GripperScrewer2.bHomingDone OR bGripperScrewer2Enable THEN	
		sHomingText:=Concat(sHomingText,'ZS2,'); END_IF	
		
	IF( NOT P10_GripperScrewer.fbGripperScrewer1CatchStation.bHomingDone AND NOT P10_GripperScrewer.fbGripperScrewer2CatchStation.bHomingDone ) OR bGripperScrewer1Enable OR bGripperScrewer2Enable THEN	
		sHomingText:=Concat(sHomingText,'CHZS,'); END_IF
			
	IF NOT P11_CapCorrectCheck.fbCapCorrectCheck.bHomingDone OR bCapCorrectCheckEnable THEN	
		sHomingText:=Concat(sHomingText,'SN,'); END_IF
		
	IF (NOT bFirstPositioningDone OR GVL.bGateRobotEnable)  THEN
		sHomingText:=Concat(sHomingText,'SZR,'); END_IF
		
	IF (NOT P13_BottleTransfer.fbBottleTransfer.bHomingDone OR bBottleTransferEnable)  THEN
		sHomingText:=Concat(sHomingText,'R,'); END_IF
		
ELSIF P00_PackML.fbPMLAuto.ePMLState = E_PMLState.ePMLState_RESETTING AND NOT bRecipeChangePositioning THEN
	
	IF VIS.bDispencersHoming AND bDispencer1Enable THEN
		sHomingText:=Concat(sHomingText,'D1,'); END_IF
		
	IF VIS.bDispencersHoming AND bDispencer2Enable THEN
		sHomingText:=Concat(sHomingText,'D2,'); END_IF
		
	IF VIS.bDispencersHoming AND bDispencer3Enable THEN
		sHomingText:=Concat(sHomingText,'D3,'); END_IF
		
	IF VIS.bDispencersHoming AND bDispencer4Enable THEN
		sHomingText:=Concat(sHomingText,'D4,'); END_IF
		
	IF VIS.bFormsDragingRightHoming AND GVL.bFormsDragingRightEnable THEN
		sHomingText:=Concat(sHomingText,'PFDP,'); END_IF

	IF VIS.bFormsDragingLeftHoming AND GVL.bFormsDragingLeftEnable THEN
		sHomingText:=Concat(sHomingText,'PFDL,'); END_IF
			
	IF VIS.bDispencersHoming THEN
		sHomingText:=Concat(sHomingText,'CHD,'); END_IF
		
	IF VIS.bWeightLiftHoming THEN	
		sHomingText:=Concat(sHomingText,'W,'); END_IF	
	
	IF VIS.bCapPuttedCheckHoming THEN	
		sHomingText:=Concat(sHomingText,'SN,'); END_IF

	IF VIS.bBottleDragingStationHoming AND GVL.bBottleDragingStationEnable THEN
		sHomingText:=Concat(sHomingText,'PFPZ,'); END_IF
		
	IF VIS.bGripperScrewerHoming THEN	
		sHomingText:=Concat(sHomingText,'ZS,'); END_IF	
		
	IF VIS.bGripperScrewerHoming THEN	
		sHomingText:=Concat(sHomingText,'CHZS,'); END_IF
		
	IF VIS.bCapCorrectCheckHoming THEN	
		sHomingText:=Concat(sHomingText,'PN,'); END_IF
		
	IF (VIS.bBottleTransferHoming)  THEN
		sHomingText:=Concat(sHomingText,'R,'); END_IF
		
	IF (VIS.bCapFeederHoming) THEN
		sHomingText:=Concat(sHomingText,'PN,'); END_IF

	
ELSE
	sHomingText:='';
END_IF




(*OBECNOSC FORMATEK***********************************************************************)
VIS.nBottleSorterPackageState_FormPresent.1					:=eBottleFeederPackageState[1].bFormPresent;

VIS.nBeforeDispencersPackageState_FormPresent.1				:=	(eBeforeDispencersPackageState[1].bFormPresent AND NOT bDosingTwoPhases)  OR (eAfterDispencer12PackageState2Phase[1].bFormPresent AND bDosingTwoPhases) ;
VIS.nBeforeDispencersPackageState_FormPresent.2				:=	(eBeforeDispencersPackageState[2].bFormPresent AND NOT bDosingTwoPhases)  OR (eAfterDispencer12PackageState2Phase[2].bFormPresent AND bDosingTwoPhases);
VIS.nBeforeDispencersPackageState_FormPresent.3				:=	(eBeforeDispencersPackageState[3].bFormPresent AND NOT bDosingTwoPhases)  OR (eBeforeDispencer34PackageState2Phase[1].bFormPresent AND bDosingTwoPhases);
VIS.nBeforeDispencersPackageState_FormPresent.4				:=	(eBeforeDispencersPackageState[4].bFormPresent AND NOT bDosingTwoPhases)  OR (eBeforeDispencer34PackageState2Phase[2].bFormPresent AND bDosingTwoPhases);
   






                                                           	
VIS.nDispencersPackageState_FormPresent.4					:=	(eDispencersPackageState[4].bFormPresent AND NOT bDosingTwoPhases) OR (eDispencer34PackageState2Phase[2].bFormPresent AND bDosingTwoPhases);
VIS.nDispencersPackageState_FormPresent.3					:=	(eDispencersPackageState[3].bFormPresent AND NOT bDosingTwoPhases) OR (eDispencer34PackageState2Phase[1].bFormPresent AND bDosingTwoPhases);
VIS.nDispencersPackageState_FormPresent.2					:=	(eDispencersPackageState[2].bFormPresent AND NOT bDosingTwoPhases) OR (eDispencer12PackageState2Phase[2].bFormPresent AND bDosingTwoPhases);
VIS.nDispencersPackageState_FormPresent.1					:=	(eDispencersPackageState[1].bFormPresent AND NOT bDosingTwoPhases) OR (eDispencer12PackageState2Phase[1].bFormPresent AND bDosingTwoPhases);
                                                              	
VIS.nAfterDispencersPackageState_FormPresent.4  			:=	(eAfterDispencersPackageState[4].bFormPresent AND NOT bDosingTwoPhases)  OR (eAfterDispencer34PackageState2Phase[2].bFormPresent AND bDosingTwoPhases);
VIS.nAfterDispencersPackageState_FormPresent.3  			:=	(eAfterDispencersPackageState[3].bFormPresent AND NOT bDosingTwoPhases)  OR (eAfterDispencer34PackageState2Phase[1].bFormPresent AND bDosingTwoPhases);
VIS.nAfterDispencersPackageState_FormPresent.2  			:=	(eAfterDispencersPackageState[2].bFormPresent AND NOT bDosingTwoPhases)  OR (eBeforeDispencer12PackageState2Phase[2].bFormPresent AND bDosingTwoPhases);
VIS.nAfterDispencersPackageState_FormPresent.1  			:=	(eAfterDispencersPackageState[1].bFormPresent AND NOT bDosingTwoPhases)  OR (eBeforeDispencer12PackageState2Phase[1].bFormPresent AND bDosingTwoPhases);
                                                              	
//VIS.nWeightPackageState_FormPresent.5  						:=	eWeightPackageState[5].bFormPresent; // nie używany, ale obecny na wizce 08.04.2022 DJA
VIS.nWeightPackageState_FormPresent.4  						:=	eWeightPackageState[4].bFormPresent;
VIS.nWeightPackageState_FormPresent.3  						:=	eWeightPackageState[3].bFormPresent;
VIS.nWeightPackageState_FormPresent.2  						:=	eWeightPackageState[2].bFormPresent;
VIS.nWeightPackageState_FormPresent.1  						:=	eWeightPackageState[1].bFormPresent;


VIS.nWeight2PackageState_FormPresent.3						:=	eWeightPackage2PhasePackageState[3].bFormPresent;  //dodane 08.04.2022 DJA
VIS.nWeight2PackageState_FormPresent.2						:=	eWeightPackage2PhasePackageState[2].bFormPresent;	//dodane 08.04.2022 DJA
VIS.nWeight2PackageState_FormPresent.1						:=	eWeightPackage2PhasePackageState[1].bFormPresent;	//dodane 08.04.2022 DJA
                                                              	
VIS.nBeforeScrewersPackageState_FormPresent.4  				:=	eBeforeScrewers2PackageState[2].bFormPresent;
VIS.nBeforeScrewersPackageState_FormPresent.3  				:=	eBeforeScrewers2PackageState[1].bFormPresent;
VIS.nBeforeScrewersPackageState_FormPresent.2  				:=	eBeforeScrewersPackageState[2].bFormPresent;
VIS.nBeforeScrewersPackageState_FormPresent.1  				:=	eBeforeScrewersPackageState[1].bFormPresent;
                                                              	
VIS.nUnderScrewerPackageState_FormPresent.2  				:=	eUnderScrewerPackageState[2].bFormPresent;
VIS.nUnderScrewerPackageState_FormPresent.1  				:=	eUnderScrewerPackageState[1].bFormPresent;
                                             				  	
VIS.nAfterScrewerPackageState_FormPresent.2  				:=	eAfterScrewerPackageState[2].bFormPresent;
VIS.nAfterScrewerPackageState_FormPresent.1  				:=	eAfterScrewerPackageState[1].bFormPresent;

VIS.nUnderCorrectCapPackageState_FormPresent.8				:=	eUnderCorrectCapPackageState[1].bFormPresent; //bylo 8
VIS.nUnderCorrectCapPackageState_FormPresent.7				:=	eUnderCorrectCapPackageState[7].bFormPresent;
VIS.nUnderCorrectCapPackageState_FormPresent.6				:=	eUnderCorrectCapPackageState[6].bFormPresent;
VIS.nUnderCorrectCapPackageState_FormPresent.5				:=	eUnderCorrectCapPackageState[5].bFormPresent;
VIS.nUnderCorrectCapPackageState_FormPresent.4				:=	eUnderCorrectCapPackageState[4].bFormPresent;
VIS.nUnderCorrectCapPackageState_FormPresent.3				:=	eUnderCorrectCapPackageState[3].bFormPresent;
VIS.nUnderCorrectCapPackageState_FormPresent.2				:=	eUnderCorrectCapPackageState[2].bFormPresent;
//VIS.nUnderCorrectCapPackageState_FormPresent.1				:=	eUnderCorrectCapPackageState[1].bFormPresent;
                                                              	
VIS.nRobotPackageState_FormPresent.2						:=	eRobotPackageState[2].bFormPresent;
VIS.nRobotPackageState_FormPresent.1						:=	eRobotPackageState[1].bFormPresent;



(*OBECNOSC BUTELEK*)
VIS.nBottleSorterPackageState_BottlePresent.1					:=eBottleFeederPackageState[1].bBottlePresent;

VIS.nBeforeDispencersPackageState_BottlePresent.4			:=	(eBeforeDispencersPackageState[4].bBottlePresent AND NOT bDosingTwoPhases) OR (eBeforeDispencer34PackageState2Phase[2].bBottlePresent AND bDosingTwoPhases); 
VIS.nBeforeDispencersPackageState_BottlePresent.3			:=	(eBeforeDispencersPackageState[3].bBottlePresent AND NOT bDosingTwoPhases) OR (eBeforeDispencer34PackageState2Phase[1].bBottlePresent AND bDosingTwoPhases); 
VIS.nBeforeDispencersPackageState_BottlePresent.2			:=	(eBeforeDispencersPackageState[2].bBottlePresent AND NOT bDosingTwoPhases) OR (eAfterDispencer12PackageState2Phase[1].bBottlePresent AND bDosingTwoPhases);
VIS.nBeforeDispencersPackageState_BottlePresent.1			:=	(eBeforeDispencersPackageState[1].bBottlePresent AND NOT bDosingTwoPhases) OR (eAfterDispencer12PackageState2Phase[2].bBottlePresent AND bDosingTwoPhases);             
                                         	
VIS.nDispencersPackageState_BottlePresent.4					:=	(eDispencersPackageState[4].bBottlePresent AND NOT bDosingTwoPhases) OR (eDispencer34PackageState2Phase[2].bBottlePresent AND bDosingTwoPhases);
VIS.nDispencersPackageState_BottlePresent.3					:=	(eDispencersPackageState[3].bBottlePresent AND NOT bDosingTwoPhases) OR (eDispencer34PackageState2Phase[1].bBottlePresent AND bDosingTwoPhases);
VIS.nDispencersPackageState_BottlePresent.2					:=	(eDispencersPackageState[2].bBottlePresent AND NOT bDosingTwoPhases) OR (eDispencer12PackageState2Phase[2].bBottlePresent AND bDosingTwoPhases);
VIS.nDispencersPackageState_BottlePresent.1					:=	(eDispencersPackageState[1].bBottlePresent AND NOT bDosingTwoPhases) OR (eDispencer12PackageState2Phase[1].bBottlePresent AND bDosingTwoPhases);
                                                       
VIS.nAfterDispencersPackageState_BottlePresent.4  			:=	(eAfterDispencersPackageState[4].bBottlePresent AND NOT bDosingTwoPhases)	OR (eAfterDispencer34PackageState2Phase[2].bBottlePresent AND bDosingTwoPhases); 
VIS.nAfterDispencersPackageState_BottlePresent.3  			:=	(eAfterDispencersPackageState[3].bBottlePresent AND NOT bDosingTwoPhases)	OR (eAfterDispencer34PackageState2Phase[1].bBottlePresent AND bDosingTwoPhases); 
VIS.nAfterDispencersPackageState_BottlePresent.2  			:=	(eAfterDispencersPackageState[2].bBottlePresent AND NOT bDosingTwoPhases)	OR (eBeforeDispencer12PackageState2Phase[2].bBottlePresent AND bDosingTwoPhases);
VIS.nAfterDispencersPackageState_BottlePresent.1  			:=	(eAfterDispencersPackageState[1].bBottlePresent AND NOT bDosingTwoPhases)	OR (eBeforeDispencer12PackageState2Phase[1].bBottlePresent AND bDosingTwoPhases);
     



                                                         	
//VIS.nWeightPackageState_BottlePresent.5  					:=	eWeightPackageState[5].bBottlePresent; // nie używany, ale obecny na wizce 08.04.2022 DJA
VIS.nWeightPackageState_BottlePresent.4  					:=	eWeightPackageState[4].bBottlePresent;
VIS.nWeightPackageState_BottlePresent.3  					:=	eWeightPackageState[3].bBottlePresent;
VIS.nWeightPackageState_BottlePresent.2  					:=	eWeightPackageState[2].bBottlePresent;
VIS.nWeightPackageState_BottlePresent.1  					:=	eWeightPackageState[1].bBottlePresent;

VIS.nWeight2PackageState_BottlePresent.3					:=	eWeightPackage2PhasePackageState[3].bBottlePresent;  //dodane 08.04.2022 DJA
VIS.nWeight2PackageState_BottlePresent.2					:=	eWeightPackage2PhasePackageState[2].bBottlePresent;	//dodane 08.04.2022 DJA
VIS.nWeight2PackageState_BottlePresent.1					:=	eWeightPackage2PhasePackageState[1].bBottlePresent;	//dodane 08.04.2022 DJA

                                                              	
VIS.nBeforeScrewersPackageState_BottlePresent.4  			:=	eBeforeScrewers2PackageState[2].bBottlePresent;
VIS.nBeforeScrewersPackageState_BottlePresent.3  			:=	eBeforeScrewers2PackageState[1].bBottlePresent;
VIS.nBeforeScrewersPackageState_BottlePresent.2  			:=	eBeforeScrewersPackageState[2].bBottlePresent;
VIS.nBeforeScrewersPackageState_BottlePresent.1  			:=	eBeforeScrewersPackageState[1].bBottlePresent;
                                                              	
VIS.nUnderScrewerPackageState_BottlePresent.2  				:=	eUnderScrewerPackageState[2].bBottlePresent;
VIS.nUnderScrewerPackageState_BottlePresent.1  				:=	eUnderScrewerPackageState[1].bBottlePresent;
                                               				  	
VIS.nAfterScrewerPackageState_BottlePresent.2  				:=	eAfterScrewerPackageState[2].bBottlePresent;
VIS.nAfterScrewerPackageState_BottlePresent.1  				:=	eAfterScrewerPackageState[1].bBottlePresent;
                                                              	
VIS.nUnderCorrectCapPackageState_BottlePresent.8			:=	eUnderCorrectCapPackageState[1].bBottlePresent; //było 8
VIS.nUnderCorrectCapPackageState_BottlePresent.7			:=	eUnderCorrectCapPackageState[7].bBottlePresent;
VIS.nUnderCorrectCapPackageState_BottlePresent.6			:=	eUnderCorrectCapPackageState[6].bBottlePresent;
VIS.nUnderCorrectCapPackageState_BottlePresent.5			:=	eUnderCorrectCapPackageState[5].bBottlePresent;
VIS.nUnderCorrectCapPackageState_BottlePresent.4			:=	eUnderCorrectCapPackageState[4].bBottlePresent;
VIS.nUnderCorrectCapPackageState_BottlePresent.3			:=	eUnderCorrectCapPackageState[3].bBottlePresent;
VIS.nUnderCorrectCapPackageState_BottlePresent.2			:=	eUnderCorrectCapPackageState[2].bBottlePresent;
///VIS.nUnderCorrectCapPackageState_BottlePresent.1			:=	eUnderCorrectCapPackageState[1].bBottlePresent;
                                                              	
VIS.nRobotPackageState_BottlePresent.2						:=	eRobotPackageState[2].bBottlePresent;
VIS.nRobotPackageState_BottlePresent.1						:=	eRobotPackageState[1].bBottlePresent;





(*WAGA OK*)
//VIS.nWeightPackageState_WeightOK.5  						:=	eWeightPackageState[5].bWeightOK; // nie używany, ale obecny na wizce 08.04.2022 DJA
VIS.nWeightPackageState_WeightOK.4  						:=	eWeightPackageState[4].bWeightOK;
VIS.nWeightPackageState_WeightOK.3  						:=	eWeightPackageState[3].bWeightOK;
VIS.nWeightPackageState_WeightOK.2  						:=	eWeightPackageState[2].bWeightOK;
VIS.nWeightPackageState_WeightOK.1  						:=	eWeightPackageState[1].bWeightOK;

VIS.nWeight2PackageState_WeightOK.3							:=	eWeightPackage2PhasePackageState[3].bWeightOK;  //dodane 08.04.2022 DJA
VIS.nWeight2PackageState_WeightOK.2							:=	eWeightPackage2PhasePackageState[2].bWeightOK;	//dodane 08.04.2022 DJA
VIS.nWeight2PackageState_WeightOK.1							:=	eWeightPackage2PhasePackageState[1].bWeightOK;	//dodane 08.04.2022 DJA


                                                          	
VIS.nBeforeScrewersPackageState_WeightOK.4  				:=	eBeforeScrewers2PackageState[2].bWeightOK;
VIS.nBeforeScrewersPackageState_WeightOK.3  				:=	eBeforeScrewers2PackageState[1].bWeightOK;
VIS.nBeforeScrewersPackageState_WeightOK.2  				:=	eBeforeScrewersPackageState[2].bWeightOK;
VIS.nBeforeScrewersPackageState_WeightOK.1  				:=	eBeforeScrewersPackageState[1].bWeightOK;
                                                              	
VIS.nUnderScrewerPackageState_WeightOK.2  					:=	eUnderScrewerPackageState[2].bWeightOK;
VIS.nUnderScrewerPackageState_WeightOK.1  					:=	eUnderScrewerPackageState[1].bWeightOK;
                                          					  	
VIS.nAfterScrewerPackageState_WeightOK.2  					:=	eAfterScrewerPackageState[2].bWeightOK;
VIS.nAfterScrewerPackageState_WeightOK.1  					:=	eAfterScrewerPackageState[1].bWeightOK;
                                                              	
VIS.nUnderCorrectCapPackageState_WeightOK.8 				:=	eUnderCorrectCapPackageState[1].bWeightOK;
VIS.nUnderCorrectCapPackageState_WeightOK.7 				:=	eUnderCorrectCapPackageState[7].bWeightOK;
VIS.nUnderCorrectCapPackageState_WeightOK.6 				:=	eUnderCorrectCapPackageState[6].bWeightOK;
VIS.nUnderCorrectCapPackageState_WeightOK.5 				:=	eUnderCorrectCapPackageState[5].bWeightOK;
VIS.nUnderCorrectCapPackageState_WeightOK.4 				:=	eUnderCorrectCapPackageState[4].bWeightOK;
VIS.nUnderCorrectCapPackageState_WeightOK.3 				:=	eUnderCorrectCapPackageState[3].bWeightOK;
VIS.nUnderCorrectCapPackageState_WeightOK.2 				:=	eUnderCorrectCapPackageState[2].bWeightOK;
//VIS.nUnderCorrectCapPackageState_WeightOK.1 				:=	eUnderCorrectCapPackageState[1].bWeightOK;
                                                              	
VIS.nRobotPackageState_WeightOK.2							:=	eRobotPackageState[2].bWeightOK;
VIS.nRobotPackageState_WeightOK.1							:=	eRobotPackageState[1].bWeightOK;
                                 							  	



(*NASADKA OK*)
VIS.nBeforeScrewersPackageState_CapOK.4  					:=	eBeforeScrewers2PackageState[2].bCapOK;//eBeforeScrewers2PackageState[2].bCapOK;
VIS.nBeforeScrewersPackageState_CapOK.3  					:=	eBeforeScrewers2PackageState[1].bCapOK;//eBeforeScrewers2PackageState[1].bCapOK;
VIS.nBeforeScrewersPackageState_CapOK.2  					:=	eBeforeScrewersPackageState[2].bCapOK;
VIS.nBeforeScrewersPackageState_CapOK.1  					:=	eBeforeScrewersPackageState[1].bCapOK;
                                                              	
VIS.nUnderScrewerPackageState_CapOK.2  						:=	eUnderScrewerPackageState[2].bCapOK;
VIS.nUnderScrewerPackageState_CapOK.1  						:=	eUnderScrewerPackageState[1].bCapOK;
                                       						  	
VIS.nAfterScrewerPackageState_CapOK.2  						:=	eAfterScrewerPackageState[2].bCapCorrectCapOn AND eAfterScrewerPackageState[2].bCapOK;
VIS.nAfterScrewerPackageState_CapOK.1  						:=	eAfterScrewerPackageState[1].bCapCorrectCapOn AND eAfterScrewerPackageState[1].bCapOK;
                                                              	
VIS.nUnderCorrectCapPackageState_CapOK.8 					:=	eUnderCorrectCapPackageState[1].bCapCorrectCapOn AND NOT eUnderCorrectCapPackageState[1].bCapCorrectNOK;
VIS.nUnderCorrectCapPackageState_CapOK.7 					:=	eUnderCorrectCapPackageState[7].bCapCorrectCapOn AND NOT eUnderCorrectCapPackageState[7].bCapCorrectNOK;
VIS.nUnderCorrectCapPackageState_CapOK.6 					:=	eUnderCorrectCapPackageState[6].bCapCorrectCapOn AND NOT eUnderCorrectCapPackageState[6].bCapCorrectNOK;
VIS.nUnderCorrectCapPackageState_CapOK.5 					:=	eUnderCorrectCapPackageState[5].bCapCorrectCapOn AND NOT eUnderCorrectCapPackageState[5].bCapCorrectNOK;
VIS.nUnderCorrectCapPackageState_CapOK.4 					:=	eUnderCorrectCapPackageState[4].bCapCorrectCapOn AND NOT eUnderCorrectCapPackageState[4].bCapCorrectNOK;
VIS.nUnderCorrectCapPackageState_CapOK.3 					:=	eUnderCorrectCapPackageState[3].bCapCorrectCapOn AND NOT eUnderCorrectCapPackageState[3].bCapCorrectNOK;
VIS.nUnderCorrectCapPackageState_CapOK.2 					:=	eUnderCorrectCapPackageState[2].bCapCorrectCapOn AND NOT eUnderCorrectCapPackageState[2].bCapCorrectNOK;
//VIS.nUnderCorrectCapPackageState_CapOK.1 					:=	eUnderCorrectCapPackageState[1].bCapCorrectCapOn AND NOT eUnderCorrectCapPackageState[1].bCapCorrectNOK;
                                                              	
VIS.nRobotPackageState_CapOK.2								:=	eRobotPackageState[2].bCapCorrectCapOn AND NOT eRobotPackageState[2].bCapCorrectNOK;
VIS.nRobotPackageState_CapOK.1								:=	eRobotPackageState[1].bCapCorrectCapOn AND NOT eRobotPackageState[1].bCapCorrectNOK;
                                                              	
                                                              	
(*ZAKRECONA*)                                                 	
VIS.nUnderScrewerPackageState_Screwed.2  					:=	eUnderScrewerPackageState[2].bCapGripperScrewed;
VIS.nUnderScrewerPackageState_Screwed.1  					:=	eUnderScrewerPackageState[1].bCapGripperScrewed;
                                         					  	
VIS.nAfterScrewerPackageState_Screwed.2  					:=	eAfterScrewerPackageState[2].bCapGripperScrewed;
VIS.nAfterScrewerPackageState_Screwed.1  					:=	eAfterScrewerPackageState[1].bCapGripperScrewed;
			                                                  	
VIS.nUnderCorrectCapPackageState_Screwed.8 					:=	eUnderCorrectCapPackageState[1].bCapGripperScrewed;
VIS.nUnderCorrectCapPackageState_Screwed.7 					:=	eUnderCorrectCapPackageState[7].bCapGripperScrewed;
VIS.nUnderCorrectCapPackageState_Screwed.6 					:=	eUnderCorrectCapPackageState[6].bCapGripperScrewed;
VIS.nUnderCorrectCapPackageState_Screwed.5 					:=	eUnderCorrectCapPackageState[5].bCapGripperScrewed;
VIS.nUnderCorrectCapPackageState_Screwed.4 					:=	eUnderCorrectCapPackageState[4].bCapGripperScrewed;
VIS.nUnderCorrectCapPackageState_Screwed.3 					:=	eUnderCorrectCapPackageState[3].bCapGripperScrewed;
VIS.nUnderCorrectCapPackageState_Screwed.2 					:=	eUnderCorrectCapPackageState[2].bCapGripperScrewed;
//VIS.nUnderCorrectCapPackageState_Screwed.1 					:=	eUnderCorrectCapPackageState[1].bCapGripperScrewed;
								
VIS.nRobotPackageState_Screwed.2							:=	eRobotPackageState[2].bCapGripperScrewed;
VIS.nRobotPackageState_Screwed.1							:=	eRobotPackageState[1].bCapGripperScrewed;

*)
END_ACTION

ACTION aCycleRegister1Phase:
eClearPackageState.nID := 0;
eClearPackageState.nCardNumber:=0;
eClearPackageState.bFormPresent := FALSE;
eClearPackageState.bBottlePresent := FALSE;
eClearPackageState.bDosingTwoPhases := FALSE;
eClearPackageState.nDispencerNr := 0;
eClearPackageState.nDispencerNrSecondPhase := 0;
eClearPackageState.tDispencingTime := T#0MS;
eClearPackageState.tDispencingTimeSecondPhase := T#0MS;
eClearPackageState.lrDoseVolumeSV := 0.0;
eClearPackageState.lrDoseVolumeCV := 0.0;
eClearPackageState.lrDoseVolumeSVSecondPhase := 0.0;
eClearPackageState.lrDoseVolumeCVSecondPhase := 0.0;
eClearPackageState.bDoseAborted := FALSE;
eClearPackageState.bWeighed := FALSE;
eClearPackageState.bWeightAborted:=FALSE;
eClearPackageState.lrWeightSV := 0.0;
eClearPackageState.lrWeightCV := 0.0;
eClearPackageState.lrWeightMeasuredCV := 0.0;
eClearPackageState.lrMinWeightCV:=0.0;
eClearPackageState.lrMaxWeightCV:=0.0;	
eClearPackageState.lrWeightDif:=0.0;			
eClearPackageState.bWeightOK := FALSE;
eClearPackageState.tWeightingTime := T#0MS;
eClearPackageState.bCapPutted := FALSE;
eClearPackageState.bCapChecked := FALSE;
eClearPackageState.bCapOK := FALSE;
eClearPackageState.bCapGripperScrewed := FALSE;
eClearPackageState.bCapGripperScrewAborted := FALSE;
eClearPackageState.tCapGripperScrewingTime := T#0MS;
eClearPackageState.bCapCorrectPutted := FALSE;
eClearPackageState.bCapCorrectChecked := FALSE;
eClearPackageState.bCapCorrectNOK := FALSE;
eClearPackageState.bCapCorrectCapOn:=FALSE;
eClearPackageState.bBottleTransferedToExit := FALSE;
eClearPackageState.bBottleTransferedToLabeler := FALSE;
bAlwaysFalse:=FALSE;

// (1) HISTORIA
fbIbFirstFormCheckFormSensor	(bIN:= 	P13_BottleTransfer.IbFirstFormCheckFormSensor,	tFilterTimeOn:=T#30MS,	tFilterTimeOff:=T#30MS);// bylo 80 i 20
ftfbIbFirstFormCheckFormSensor	(CLK:=	fbIbFirstFormCheckFormSensor.bOUT, 				Q=>);
rtfbIbFirstFormCheckFormSensor	(CLK:=	fbIbFirstFormCheckFormSensor.bOUT,				Q=>);
fbIbSecondFormCheckFormSensor	(bIN:= 	P13_BottleTransfer.IbSecondFormCheckFormSensor,	tFilterTimeOn:=T#30MS,	tFilterTimeOff:=T#30MS);
rtfbIbSecondFormCheckFormSensor	(CLK:=	fbIbSecondFormCheckFormSensor.bOUT, 			Q=>);
ftfbIbSecondFormCheckFormSensor	(CLK:=	fbIbSecondFormCheckFormSensor.bOUT, 			Q=>);


// (0) Kasowanie formatek za robotem
// BOOL ustawiany przy nastepnym ruchu robota
bRFIDClearAfterRobot;					
iRFIDClearNr1AfterRobot;	
iRFIDClearNr2AfterRobot;
rtiBottleTransferCase2(CLK:=P00_PackML.iBottleTransferCase	=	2,		Q=>);
IF	rtiBottleTransferCase2.Q	THEN
	IF P00_PackML.nCounterFormsToLoad = 2 THEN
		iRFIDClearNr1AfterRobot	:=	ULINT_TO_INT(eRobotPackageState[1].nCardNumber);
		iRFIDClearNr2AfterRobot	:=	ULINT_TO_INT(eRobotPackageState[2].nCardNumber);		
	ELSIF P00_PackML.nCounterFormsToLoad = 1 THEN
		iRFIDClearNr1AfterRobot	:=	ULINT_TO_INT(eRobotPackageState[1].nCardNumber);
		iRFIDClearNr2AfterRobot	:=	0;	
	END_IF
END_IF
IF bRFIDClearAfterRobot THEN 
	FOR i:=1 TO 100 DO	
		IF iRFIDClearNr1AfterRobot > 0 THEN	{warning 'tutaj zmienić na dwa FORy i EXITy'}
			IF eRFID[i].nCardNumber = INT_TO_ULINT(iRFIDClearNr1AfterRobot) THEN
				eRFID[i]						:=	eClearPackageState;
				eRFID[i].bFormPresent			:= TRUE; // wprowadzona zmiana do testów 
				iRFIDClearNr1AfterRobot			:= 0;
				iRFIDClearNr1AfterRobotCount	:=	iRFIDClearNr1AfterRobotCount	+	1;
			END_IF
		END_IF
		IF iRFIDClearNr2AfterRobot > 0 THEN
			IF eRFID[i].nCardNumber = INT_TO_ULINT(iRFIDClearNr2AfterRobot) THEN
				eRFID[i]						:=	eClearPackageState;
				eRFID[i].bFormPresent			:= TRUE;  // Wprowadzona zmiana do testów
				iRFIDClearNr2AfterRobot			:= 0;
				
				iRFIDClearNr2AfterRobotCount	:=	iRFIDClearNr2AfterRobotCount	+	1;
			END_IF
		END_IF		
		IF 	iRFIDClearNr1AfterRobot = 0 AND iRFIDClearNr2AfterRobot = 0 THEN
			bRFIDClearAfterRobot	:=	FALSE;
		END_IF
	END_FOR;
END_IF



IF ftfbIbFirstFormCheckFormSensor.Q THEN
	
	FOR i := 999 TO 2 BY -1 DO		
		eHistoryPackageState[i] := eHistoryPackageState[i-1];
	END_FOR		
	
	FOR i:=1 TO 100 DO	
	
		IF eRobotPackageState[1].nCardNumber=eRFID[i].nCardNumber THEN
			eRFID[i]		:=	eRobotPackageState[1];
			EXIT;
		END_IF;
	
	END_FOR;
	
	eHistoryPackageState[1]	:=	eRobotPackageState[1];
	eRobotPackageState[1]	:=	eClearPackageState; // dodane na testy
	nCheckRobotDone			:=	nCheckRobotDone+1;
	
END_IF

IF bResetStates THEN
	eRobotPackageState[1]:=eClearPackageState;
	eRobotPackageState[2]:=eClearPackageState;
	eRobotTempState[1]:=eClearPackageState;// dodane na testy 31.05
END_IF

IF nFormCounter = 1000 OR bResetHistory THEN 
	FOR i := 1 TO 1000 DO
		eHistoryPackageState[i]:=eClearPackageState;
	END_FOR
	
	nFormCounter := 0 ;
	nID := 0;
END_IF


// (2) PRZESUWANIE POD ROBOTEM
IF rtfbIbFirstFormCheckFormSensor.Q THEN
	eRobotPackageState[1]				:= eRobotTempState[1];
	eRobotTempState[1]					:= eClearPackageState;
END_IF

IF  ftfbIbSecondFormCheckFormSensor.Q THEN
	eRobotTempState[1]					:=	eRobotPackageState[2];
	eRobotPackageState[2]				:=	eClearPackageState;
END_IF

IF rtfbIbSecondFormCheckFormSensor.Q THEN
	eRobotPackageState[2].bFormPresent	:=	TRUE;
END_IF

// (3) Przesuwanie formatek zza zakrecarek pod sprwadzanie nakretek
//Przesuwanie formatek spod sprawdzania zakretek na robota
//Usuwanie rejestru bo jest nieuzywant	
//eUnderCorrectCapPackageState[1]		:=	eClearPackageState;	
eUnderCorrectCapPackageState[2]			:=	eClearPackageState;	
eUnderCorrectCapPackageState[3]			:=	eClearPackageState;	
eUnderCorrectCapPackageState[4]			:=	eClearPackageState;	
eUnderCorrectCapPackageState[5]			:=	eClearPackageState;	
eUnderCorrectCapPackageState[6]			:=	eClearPackageState;		
eUnderCorrectCapPackageState[7]			:=	eClearPackageState;		
eUnderCorrectCapPackageState[8]			:=	eClearPackageState;									//bylo 400ms?
fbIbCapCorrectCheckFormSensor			(bIN:= 	P11_CapCorrectCheck.IbCapCorrectCheckFormSensor,	tFilterTimeOn:=T#10MS,	tFilterTimeOff:=T#0MS); //BYŁO 20ms
rtfbIbCapCorrectCheckFormSensor			(CLK:=	fbIbCapCorrectCheckFormSensor.bOUT, 					Q=>); // dd do testów
ftfbIbCapCorrectCheckFormSensor			(CLK:=	fbIbCapCorrectCheckFormSensor.bOUT, 					Q=>);

//Czujnik przesuwania rejestru za zakręcarką
fbIbCapCorrectCheckAfterScrewerFormSensor (bIN:= 	P11_CapCorrectCheck.IbCapCorrectCheckAfterScrewerFormSensor,	tFilterTimeOn:=T#40MS,	tFilterTimeOff:=T#0MS); //BYŁO 20ms
ftfbIbCapCorrectCheckAfterScrewerFormSensor(CLK:=fbIbCapCorrectCheckAfterScrewerFormSensor.bOUT);

IF rtfbIbCapCorrectCheckFormSensor.Q AND NOT eUnderCorrectCapPackageState[1].bFormPresent THEN  			//dd do testów USUNAĆ
	eUnderCorrectCapPackageState[1].bFormPresent  :=	TRUE;  												//dd do testów USUNAĆ
	iTestCCC2	:=	iTestCCC2	+	1;																		//dd do testów USUNAĆ
END_IF  																								

IF 	ftfbIbCapCorrectCheckFormSensor.Q THEN
	eUnderCorrectCapPackageState[1]	:=	eClearPackageState;
	iTestCCC1	:=	iTestCCC1	+	1;
END_IF

fbMRCorrectCapPackageState(
						bFirstCycle:= GVL.bFirstCycle,
						bTrigger:=(*ftfbIbCapCorrectCheckFormSensor.Q*)ftfbIbCapCorrectCheckAfterScrewerFormSensor.Q,
						tTriggerFilterTimeOn:=T#0MS,
						tTriggerFilterTimeOff:=T#0MS,
						bTriggerBottle:=FALSE,
						bWithBottleControl:=FALSE,
						bWithCapControl:=FALSE,
						bWithFormControlTrigerCounter:=FALSE,
						bMoveOnlyToLastExitRegister:=FALSE,
						bRotateEntranceRegisterBefore:=FALSE,
						bNoKeepTryingMove:=TRUE,
						bTriggerCap:=FALSE,
						bReset:=bResetStates,
						iEntranceArrayElements:=2,
						iExitArrayElements:=8,
						bInvertWriting:=FALSE,
						eClearPackageState:=eClearPackageState,
						bTriggerCounter:=bMRCapCorrect,
						eEntranceState:=eAfterScrewerPackageState,
						//eExitState:=eUnderCorrectCapPackageState, //dd do testów USUNAĆ
						eExitState:=eUnderCorrectCapPackageStateTemp,						
						bKeepTryingMove:=bKeepTryingMove1,
						bError=>,
						iError=>,
						bTriggerDone=>,
						bTriggerFilteredOUT=>);			

eUnderCorrectCapPackageStateTemp[1]:= eClearPackageState; //dd do testów USUNAĆ
eUnderCorrectCapPackageStateTemp[2]:= eClearPackageState;//dd do testów USUNAĆ 
						
// (4) Przesuwanie formatek spod zakrecearek za zakrecarki  
//rtfbFormsDragingPneumaticStationDragging(CLK:=P10_GripperScrewer.fbGripperScrewersDragStation.eRunningState = E_DragStationState.eDraging);
rtfbFormsDragingPneumaticStationDragging(CLK:=P10_GripperScrewer.fbGripperScrewersDragStation.eRunningState = E_DragStationState.eDraging AND P10_GripperScrewer.fbGripperScrewersDragStation.lrActualDragPosition>80);

IF rtfbFormsDragingPneumaticStationDragging.Q THEN
	eAfterScrewerPackageState[1]		:=	eUnderScrewerPackageState[1];
	eAfterScrewerPackageState[2]		:=	eUnderScrewerPackageState[2];
	eUnderScrewerPackageState[1]		:=	eClearPackageState;
	eUnderScrewerPackageState[2]		:=	eClearPackageState;
END_IF

								
// (5) Przesuwanie formatek sprzed zakrecarek na zakrecarki
IF rtfbFormsDragingPneumaticStationDragging.Q THEN
	eUnderScrewerPackageState[1]		:=	eBeforeScrewersPackageState[1];
	eBeforeScrewersPackageState[1]		:=	eClearPackageState;
	eUnderScrewerPackageState[2]		:=	eBeforeScrewers2PackageState[1];
	eBeforeScrewers2PackageState[1]		:=	eClearPackageState;
END_IF

// (6) Przesuwanie formatek zza sprawdzania zalozenia na przed zakrecarki
fbIbScrewerThirdFormCheckFormSensor			(bIN:= 	P10_GripperScrewer.IbGripperScrewersThirdFormCheckFormSensor,		tFilterTimeOn:=T#30MS,	tFilterTimeOff:=T#30MS); //BYŁO 20ms
ftfbIbScrewerThirdFormCheckFormSensor		(CLK:=	fbIbScrewerThirdFormCheckFormSensor.bOUT, 			Q=>);
rtfbIbScrewerThirdFormCheckFormSensor		(CLK:=	fbIbScrewerThirdFormCheckFormSensor.bOUT, 			Q=>);
bTrendIbThirdFormCheckFormSensor:=P10_GripperScrewer.IbGripperScrewersThirdFormCheckFormSensor; 
bTrendFilteredIbThirdFormCheckFormSensor:=ftfbIbScrewerThirdFormCheckFormSensor.Q;
ftbMRBeforeScrewer2Block 					(CLK:=	bMRBeforeScrewer2Block,								Q=>);
tofftbMRBeforeScrewer2Block					(IN:=	ftbMRBeforeScrewer2Block.Q,							PT:=T#1100MS);//bylo 350		//  bylo 1000			


// Ustawianie blokady dla ruchu tylko w jedną stronę siłownika
IF ( P10_GripperScrewer.fbGripperScrewersDragStation.eRunningState = E_DragStationState.eDraging )
	AND NOT bMRBeforeScrewer2Block AND NOT tofftbMRBeforeScrewer2Block.Q THEN
	bMRBeforeScrewer2Block := TRUE;
END_IF

//IF bMRBeforeScrewer2Block AND P00_PackML.tonGripperScrewerDragMiddleSensor.Q THEN
IF bMRBeforeScrewer2Block AND P10_GripperScrewer.fbGripperScrewersDragStation.eRunningState = E_DragStationState.eDraging AND P10_GripperScrewer.fbGripperScrewersDragStation.lrActualDragPosition>90 THEN	
	bMRBeforeScrewer2Block := FALSE;
END_IF


//(6)
fbMRBeforeScrewer2PackageState(
                        bFirstCycle:= GVL.bFirstCycle,
                        bTrigger:=ftfbIbScrewerThirdFormCheckFormSensor.Q AND NOT bMRBeforeScrewer2Block,
                        tTriggerFilterTimeOn:=T#0MS,
                        tTriggerFilterTimeOff:=T#0MS,
                        bTriggerBottle:=FALSE,
                        bWithBottleControl:=FALSE,
                        bWithCapControl:=FALSE,
                        bWithFormControlTrigerCounter:=FALSE,
                        bRotateEntranceRegisterBefore:=FALSE,
                        bNoKeepTryingMove:=TRUE,
                        bTriggerCap:=,
                        bReset:=bResetStates,
                        iEntranceArrayElements:=2,
                        iExitArrayElements:=2,
                        bInvertWriting:=FALSE,
                        eClearPackageState:=eClearPackageState,
                        bTriggerCounter:=bMRFormInCap,
                        eEntranceState:=eBeforeScrewers2PackageState,
                        eExitState:=eBeforeScrewersPackageState,
                        bKeepTryingMove:=bKeepTryingMove2,
                        bError=>,
                        iError=>,
                        bTriggerDone=>,
                        bTriggerFilteredOUT=>);   										

// (6) A - Dodatkowe przesuniecie na zboczne narastajace
IF rtfbIbScrewerThirdFormCheckFormSensor.Q AND NOT eBeforeScrewers2PackageState[1].bFormPresent THEN
	eBeforeScrewers2PackageState[1] := eBeforeScrewers2PackageState[2];
	eBeforeScrewers2PackageState[2] := eClearPackageState;
END_IF

						
//(7) Przesuwanie formatek spod sprawdzania zalozenia na przed zakrecarki
fbIbCapPuttedCheckFormSensor		(bIN:= 	P09_CapPuttedCheck.IbCapPuttedCheckFormSensor,		tFilterTimeOn:=T#30MS,	tFilterTimeOff:=T#30MS); //Było 20ms
fbIbCapPuttedCheckFormSensorv2		(bIN:= 	P09_CapPuttedCheck.IbCapPuttedCheckFormSensor,		tFilterTimeOn:=T#30MS,	tFilterTimeOff:=T#30MS); //Było 20ms
ftfbIbCapPuttedCheckFormSensor		(CLK:=	fbIbCapPuttedCheckFormSensorv2.bOUT, 					Q=>);


IF ftfbIbCapPuttedCheckFormSensor.Q THEN
	iftfbIbCapPuttedCheckFormSensor := iftfbIbCapPuttedCheckFormSensor+1;
END_IF


bBitTestOn:=TRUE;


fbMRBeforeScrewerPackageState(
                        bFirstCycle:= GVL.bFirstCycle,
                        bTrigger:= ftfbIbCapPuttedCheckFormSensor.Q,
                        tTriggerFilterTimeOn:=T#0MS,
                        tTriggerFilterTimeOff:=T#0MS,
                        bWithCapControl:=TRUE,
                      	bNoKeepTryingMove:=TRUE,
                        bTriggerCap:=P09_CapPuttedCheck.eCapPuttedCheckRunningState = E_CheckerState.eCapOK,
                        bReset:=bResetStates,
                        iEntranceArrayElements:=1,
                        iExitArrayElements:=2,
                        eClearPackageState:=eClearPackageState,
                        eEntranceState:=eBeforeCapControlPackageState,
                        eExitState:=eBeforeScrewers2PackageState,
                        bKeepTryingMove:=bKeepTryingMove3,
						bRFIDReaded:=bRFIDSBeforeScrewerWriteToRegister(*bBitTestOn*), // Ustawiany jeżeli Dane z tablicy RFID zostały wpisane do zwykłego rejestru
                        iBottleWithoutCap:=iCapFeederCheckCountNOK,
						bError=>,
                        iError=>,
                        bTriggerDone=>,
                        bTriggerFilteredOUT=>);   
				


// --------------------------------------

aCycleRegisterROPP();

// (7,5-7,9) Przesuwanie pod sorterem nasadek

aCycleRegisterCapSorter();

// --------------------------------------
		
// (8) Przesuwanie formatek z wagi w kosmos				

eTempState1[1]:=eClearPackageState;
eTempState1[2]:=eClearPackageState;
eTempState1[3]:=eClearPackageState;
fbIbWeight1FormSensor			(bIN:= 	P05_Weight.IbWeight1FormSensor,		tFilterTimeOn:=T#40MS,	tFilterTimeOff:=T#40MS); //bylo 20 i 40
ftfbIbWeight1FormSensor			(CLK:=	fbIbWeight1FormSensor.bOUT, 		Q=>);		
fbMRAfterWeightPackageState(
						bFirstCycle:= GVL.bFirstCycle,
						bTrigger:=ftfbIbWeight1FormSensor.Q,
						tTriggerFilterTimeOn:=T#0MS,
						tTriggerFilterTimeOff:=T#0MS,
						bTriggerBottle:=FALSE,
						bWithBottleControl:=FALSE,
						bWithCapControl:=FALSE,
						bWithFormControlTrigerCounter:=FALSE,
						bMoveOnlyToLastExitRegister:=FALSE,
						bRotateEntranceRegisterBefore:=FALSE,
						bNoKeepTryingMove:=FALSE,
						bTriggerCap:=FALSE,
						bReset:=bResetStates,
						iEntranceArrayElements:=4,
						iExitArrayElements:=4,
						bInvertWriting:=FALSE,
						eClearPackageState:=eClearPackageState,
						bTriggerCounter:=bMRFormExitWeight,
						eEntranceState:=eWeightPackageState,
						eExitState:=eTempState1,
						bKeepTryingMove:=bKeepTryingMove4,
						bError=>,
						iError=>,
						bTriggerDone=>,
						bTriggerFilteredOUT=>);				
						
// (9) Przesuwanie formatek zza dozownikow na wage
fbIbWeight4FormSensor			(bIN:= 	P05_Weight.IbWeight4FormSensor,		tFilterTimeOn:=T#70MS,	tFilterTimeOff:=T#70MS); //BYLO 40 I 40
//fbIbWeight4FormSensor			(bIN:= 	P00_ReadRFIDCard.bReadedCardAfterDispencers,		tFilterTimeOn:=T#40MS,	tFilterTimeOff:=T#40MS); //BYLO 20 I 20
ftIbWeight4FormSensor			(CLK:=	fbIbWeight4FormSensor.bOUT, 		Q=>);	
fbMRWeightPackageState(
						bFirstCycle:= GVL.bFirstCycle,
						bTrigger:=fbIbWeight4FormSensor.bOUT,//P05_Weight.IbWeight4FormSensor, 
						tTriggerFilterTimeOn:=T#100MS,
						tTriggerFilterTimeOff:=T#20MS,
						bTriggerBottle:=FALSE,
						bWithBottleControl:=FALSE,
						bWithCapControl:=FALSE,
						bWithFormControlTrigerCounter:=FALSE,
						bMoveOnlyToLastExitRegister:=FALSE,
						bRotateEntranceRegisterBefore:=FALSE,
						bNoKeepTryingMove:=FALSE,
						bTriggerCap:=FALSE,
						bReset:=bResetStates,
						iEntranceArrayElements:=4,
						iExitArrayElements:=4,
						bInvertWriting:=FALSE,
						eClearPackageState:=eClearPackageState,
						bTriggerCounter:=bTemp,
						eEntranceState:=eAfterDispencersPackageState,
						eExitState:=eWeightPackageState,
						bKeepTryingMove:=bKeepTryingMove5,
						bError=>,
						iError=>,
						bTriggerDone=>,
						bTriggerFilteredOUT=>);		

// (10) Przesuwanie z dozownikow za dozowniki

fbMRAfterDispencerPackageState(
						bFirstCycle:= GVL.bFirstCycle,
						//bTrigger:=P02_Dispencers.fbDispencersDragRightStation.lrActualDragPosition>=130,
						bTrigger:=P00_PackML.tonDispencersDragLeftMiddleSensor.Q, {warning 'Przeciaganie - TON zamiast pozycji'}
						tTriggerFilterTimeOn:=T#0MS,
						tTriggerFilterTimeOff:=T#0MS,
						bInvertWriting:=FALSE,
						bTriggerBottle:=FALSE,
						iEntrenceArrayElements:=4,
						iExitArrayElements:=4,
						bWithFormControlTrigerCounter:=FALSE,
						bMoveOnlyIfFormPresent:=FALSE,
						bMoveOnlyToLastExitRegister:=FALSE,
						bMoveOnlyToLastRegister:=FALSE,
						bNoKeepTryingMove:=FALSE,
						bReset:=bResetStates,
						eClearPackageState:=eClearPackageState,
						bRotateEntranceRegisterBefore:=FALSE,
						bTriggerCounter:=bMRFormExitDispencer,
						eEntranceState:=eDispencersPackageState,
						eExitState:=eAfterDispencersPackageState,
						bKeepTryingMove:=bKeepTryingMove6,
						bError=>,
						iError=>,
						bTriggerDone=>,
						bTriggerFilteredOUT=>);	

// (11) Przesuwanie sprzed dozownikow na dozowniki
fbMRDispencerPackageState(
						bFirstCycle:= GVL.bFirstCycle,
						//bTrigger:=P02_Dispencers.fbDispencersDragRightStation.lrActualDragPosition>=130,
						bTrigger:=P00_PackML.tonDispencersDragLeftMiddleSensor.Q, {warning 'Przeciaganie - TON zamiast pozycji'}						
						tTriggerFilterTimeOn:=T#0MS,
						tTriggerFilterTimeOff:=T#0MS,
						bInvertWriting:=FALSE,
						bTriggerBottle:=FALSE,
						iEntrenceArrayElements:=4,
						iExitArrayElements:=4,
						bWithFormControlTrigerCounter:=FALSE,
						bMoveOnlyIfFormPresent:=FALSE,
						bMoveOnlyToLastExitRegister:=FALSE,
						bMoveOnlyToLastRegister:=FALSE,
						bNoKeepTryingMove:=FALSE,
						bReset:=bResetStates,
						eClearPackageState:=eClearPackageState,
						bRotateEntranceRegisterBefore:=FALSE,
						bTriggerCounter:=bMRFormDispencer,
						eEntranceState:=eBeforeDispencersPackageState,
						eExitState:=eDispencersPackageState,
						bKeepTryingMove:=bKeepTryingMove7,
						bError=>,
						iError=>,
						bTriggerDone=>,
						bTriggerFilteredOUT=>);		
					
// (12) Przesuwanie formatek sprzed szlabanu rpzed dozowniki

fbFilteredFormsSensorGate(bIn:=IbFormCheckFormSensor,	tFilterTimeOn:=T#30MS,	tFilterTimeOff:=T#20MS);					
fbMRBeforeDispencersPackageStateNew(
						bFirstCycle:= GVL.bFirstCycle,
						{warning ''}
						bTrigger:=(*fbFilteredFormsSensorGate.bOUT*)bFormatSensor,
						tTriggerFilterTimeOn:=T#0MS,
						tTriggerFilterTimeOff:=T#0MS,
						{warning 'Add filtered value 2023/06/16'}
						bTriggerBottle:=bBottleSensor (*MAIN.IbBottleInFormCheckBottleSensor*) OR VIS.bSimulation,
						bWithBottleControl:=TRUE,
						bWithCapControl:=FALSE,
						bWithFormControlTrigerCounter:=FALSE,
						bMoveOnlyToLastExitRegister:=FALSE,
						bRotateEntranceRegisterBefore:=FALSE,
						bNoKeepTryingMove:=TRUE,
						bTriggerCap:=,
						bReset:=bResetStates,
						iEntranceArrayElements:=1,
						iExitArrayElements:=4,
						bInvertWriting:=FALSE,
						eClearPackageState:=eClearPackageState,
						bTriggerCounter:=bMRFormExitGate1,
						eEntranceState:=eBeforeGatePackageState,
						eExitState:=eBeforeDispencersPackageState,
						bKeepTryingMove:=bKeepTryingMove8,
						bError=>,
						iError=>,
						bTriggerDone=>,
						bTriggerFilteredOUT=>);	
						
// Przesuwanie formatek spod podjanika butelek w kosmos
eTempState2[1]:=eClearPackageState;
eTempState2[2]:=eClearPackageState;
eTempState2[3]:=eClearPackageState;
fbIbBottleFeederFormPresent(bIn:=P01_BottleFeeder.IbBottleFeederFormGateBeforeSensor,	tFilterTimeOn:=T#20MS,	tFilterTimeOff:=T#20MS);					
ftfbIbBottleFeederFormPresent(CLK:=fbIbBottleFeederFormPresent.bOUT);

						
aSetIDBottle();						
						
//Pierwszy cykl, zeby na poczatek nie wykrywalo zbocza opadajacego				
bFirstCycle:=TRUE;		
GVL.bResetStates:=FALSE;


(**** Zapisywanie RFID  ***)

a2RFID();

(**** Koniec zapisywania RFID  ***)
END_ACTION

ACTION aCycleRegister1PhaseLidFeederOrWick:
eClearPackageState.nID := 0;
eClearPackageState.nCardNumber:=0;
eClearPackageState.bFormPresent := FALSE;
eClearPackageState.bBottlePresent := FALSE;
eClearPackageState.bDosingTwoPhases := FALSE;
eClearPackageState.nDispencerNr := 0;
eClearPackageState.nDispencerNrSecondPhase := 0;
eClearPackageState.tDispencingTime := T#0MS;
eClearPackageState.tDispencingTimeSecondPhase := T#0MS;
eClearPackageState.lrDoseVolumeSV := 0.0;
eClearPackageState.lrDoseVolumeCV := 0.0;
eClearPackageState.lrDoseVolumeSVSecondPhase := 0.0;
eClearPackageState.lrDoseVolumeCVSecondPhase := 0.0;
eClearPackageState.bDoseAborted := FALSE;
eClearPackageState.bWeighed := FALSE;
eClearPackageState.bWeightAborted:=FALSE;
eClearPackageState.lrWeightSV := 0.0;
eClearPackageState.lrWeightCV := 0.0;
eClearPackageState.lrWeightMeasuredCV := 0.0;
eClearPackageState.lrMinWeightCV:=0.0;
eClearPackageState.lrMaxWeightCV:=0.0;	
eClearPackageState.lrWeightDif:=0.0;			
eClearPackageState.bWeightOK := FALSE;
eClearPackageState.tWeightingTime := T#0MS;
eClearPackageState.bCapPutted := FALSE;
eClearPackageState.bCapChecked := FALSE;
eClearPackageState.bCapOK := FALSE;
eClearPackageState.bCapGripperScrewed := FALSE;
eClearPackageState.bCapGripperScrewAborted := FALSE;
eClearPackageState.tCapGripperScrewingTime := T#0MS;
eClearPackageState.bCapCorrectPutted := FALSE;
eClearPackageState.bCapCorrectChecked := FALSE;
eClearPackageState.bCapCorrectNOK := FALSE;
eClearPackageState.bCapCorrectCapOn:=FALSE;
eClearPackageState.bBottleTransferedToExit := FALSE;
eClearPackageState.bBottleTransferedToLabeler := FALSE;
bAlwaysFalse:=FALSE;

// (1) HISTORIA
fbIbFirstFormCheckFormSensor	(bIN:= 	P13_BottleTransfer.IbFirstFormCheckFormSensor,	tFilterTimeOn:=T#30MS,	tFilterTimeOff:=T#30MS);// bylo 80 i 20
ftfbIbFirstFormCheckFormSensor	(CLK:=	fbIbFirstFormCheckFormSensor.bOUT, 				Q=>);
rtfbIbFirstFormCheckFormSensor	(CLK:=	fbIbFirstFormCheckFormSensor.bOUT,				Q=>);
fbIbSecondFormCheckFormSensor	(bIN:= 	P13_BottleTransfer.IbSecondFormCheckFormSensor,	tFilterTimeOn:=T#30MS,	tFilterTimeOff:=T#30MS);
rtfbIbSecondFormCheckFormSensor	(CLK:=	fbIbSecondFormCheckFormSensor.bOUT, 			Q=>);
ftfbIbSecondFormCheckFormSensor	(CLK:=	fbIbSecondFormCheckFormSensor.bOUT, 			Q=>);


// (0) Kasowanie formatek za robotem
// BOOL ustawiany przy nastepnym ruchu robota
bRFIDClearAfterRobot;					
iRFIDClearNr1AfterRobot;	
iRFIDClearNr2AfterRobot;
rtiBottleTransferCase2(CLK:=P00_PackML.iBottleTransferCase	=	2,		Q=>);
IF	rtiBottleTransferCase2.Q	THEN
	IF P00_PackML.nCounterFormsToLoad = 2 THEN
		iRFIDClearNr1AfterRobot	:=	ULINT_TO_INT(eRobotPackageState[1].nCardNumber);
		iRFIDClearNr2AfterRobot	:=	ULINT_TO_INT(eRobotPackageState[2].nCardNumber);		
	ELSIF P00_PackML.nCounterFormsToLoad = 1 THEN
		iRFIDClearNr1AfterRobot	:=	ULINT_TO_INT(eRobotPackageState[1].nCardNumber);
		iRFIDClearNr2AfterRobot	:=	0;	
	END_IF
END_IF
IF bRFIDClearAfterRobot THEN 
	FOR i:=1 TO 100 DO	
		IF iRFIDClearNr1AfterRobot > 0 THEN	{warning 'tutaj zmienić na dwa FORy i EXITy'}
			IF eRFID[i].nCardNumber = INT_TO_ULINT(iRFIDClearNr1AfterRobot) THEN
				eRFID[i]						:=	eClearPackageState;
				eRFID[i].bFormPresent			:= TRUE; // wprowadzona zmiana do testów 
				iRFIDClearNr1AfterRobot			:= 0;
				iRFIDClearNr1AfterRobotCount	:=	iRFIDClearNr1AfterRobotCount	+	1;
			END_IF
		END_IF
		IF iRFIDClearNr2AfterRobot > 0 THEN
			IF eRFID[i].nCardNumber = INT_TO_ULINT(iRFIDClearNr2AfterRobot) THEN
				eRFID[i]						:=	eClearPackageState;
				eRFID[i].bFormPresent			:= TRUE;  // Wprowadzona zmiana do testów
				iRFIDClearNr2AfterRobot			:= 0;
				
				iRFIDClearNr2AfterRobotCount	:=	iRFIDClearNr2AfterRobotCount	+	1;
			END_IF
		END_IF		
		IF 	iRFIDClearNr1AfterRobot = 0 AND iRFIDClearNr2AfterRobot = 0 THEN
			bRFIDClearAfterRobot	:=	FALSE;
		END_IF
	END_FOR;
END_IF



IF ftfbIbFirstFormCheckFormSensor.Q THEN
	
	FOR i := 999 TO 2 BY -1 DO		
		eHistoryPackageState[i] := eHistoryPackageState[i-1];
	END_FOR		
	
	FOR i:=1 TO 100 DO	
	
		IF eRobotPackageState[1].nCardNumber=eRFID[i].nCardNumber THEN
			eRFID[i]		:=	eRobotPackageState[1];
			EXIT;
		END_IF;
	
	END_FOR;
	
	eHistoryPackageState[1]	:=	eRobotPackageState[1];
	eRobotPackageState[1]	:=	eClearPackageState; // dodane na testy
	nCheckRobotDone			:=	nCheckRobotDone+1;
	
END_IF

IF bResetStates THEN
	eRobotPackageState[1]:=eClearPackageState;
	eRobotPackageState[2]:=eClearPackageState;
	eRobotTempState[1]:=eClearPackageState;// dodane na testy 31.05
END_IF

IF nFormCounter = 1000 OR bResetHistory THEN 
	FOR i := 1 TO 1000 DO
		eHistoryPackageState[i]:=eClearPackageState;
	END_FOR
	
	nFormCounter := 0 ;
	nID := 0;
END_IF


// (2) PRZESUWANIE POD ROBOTEM
IF rtfbIbFirstFormCheckFormSensor.Q THEN
	eRobotPackageState[1]				:= eRobotTempState[1];
	eRobotTempState[1]					:= eClearPackageState;
END_IF

IF  ftfbIbSecondFormCheckFormSensor.Q THEN
	eRobotTempState[1]					:=	eRobotPackageState[2];
	eRobotPackageState[2]				:=	eClearPackageState;
END_IF

IF rtfbIbSecondFormCheckFormSensor.Q THEN
	eRobotPackageState[2].bFormPresent	:=	TRUE;
END_IF

// (3) Przesuwanie formatek zza zakrecarek pod sprwadzanie nakretek
//Przesuwanie formatek spod sprawdzania zakretek na robota
//Usuwanie rejestru bo jest nieuzywant	
//eUnderCorrectCapPackageState[1]		:=	eClearPackageState;	
eUnderCorrectCapPackageState[2]			:=	eClearPackageState;	
eUnderCorrectCapPackageState[3]			:=	eClearPackageState;	
eUnderCorrectCapPackageState[4]			:=	eClearPackageState;	
eUnderCorrectCapPackageState[5]			:=	eClearPackageState;	
eUnderCorrectCapPackageState[6]			:=	eClearPackageState;		
eUnderCorrectCapPackageState[7]			:=	eClearPackageState;		
eUnderCorrectCapPackageState[8]			:=	eClearPackageState;									//bylo 400ms?
fbIbCapCorrectCheckFormSensor			(bIN:= 	P11_CapCorrectCheck.IbCapCorrectCheckFormSensor,	tFilterTimeOn:=T#10MS,	tFilterTimeOff:=T#0MS); //BYŁO 20ms
rtfbIbCapCorrectCheckFormSensor			(CLK:=	fbIbCapCorrectCheckFormSensor.bOUT, 					Q=>); // dd do testów
ftfbIbCapCorrectCheckFormSensor			(CLK:=	fbIbCapCorrectCheckFormSensor.bOUT, 					Q=>);

//Czujnik przesuwania rejestru za zakręcarką
fbIbCapCorrectCheckAfterScrewerFormSensor (bIN:= 	P11_CapCorrectCheck.IbCapCorrectCheckAfterScrewerFormSensor,	tFilterTimeOn:=T#40MS,	tFilterTimeOff:=T#0MS); //BYŁO 20ms
ftfbIbCapCorrectCheckAfterScrewerFormSensor(CLK:=fbIbCapCorrectCheckAfterScrewerFormSensor.bOUT);

IF rtfbIbCapCorrectCheckFormSensor.Q AND NOT eUnderCorrectCapPackageState[1].bFormPresent THEN  			//dd do testów USUNAĆ
	eUnderCorrectCapPackageState[1].bFormPresent  :=	TRUE;  												//dd do testów USUNAĆ
	iTestCCC2	:=	iTestCCC2	+	1;																		//dd do testów USUNAĆ
END_IF  																								

IF 	ftfbIbCapCorrectCheckFormSensor.Q THEN
	eUnderCorrectCapPackageState[1]	:=	eClearPackageState;
	iTestCCC1	:=	iTestCCC1	+	1;
END_IF

fbMRCorrectCapPackageState(
						bFirstCycle:= GVL.bFirstCycle,
						bTrigger:=(*ftfbIbCapCorrectCheckFormSensor.Q*)ftfbIbCapCorrectCheckAfterScrewerFormSensor.Q,
						tTriggerFilterTimeOn:=T#0MS,
						tTriggerFilterTimeOff:=T#0MS,
						bTriggerBottle:=FALSE,
						bWithBottleControl:=FALSE,
						bWithCapControl:=FALSE,
						bWithFormControlTrigerCounter:=FALSE,
						bMoveOnlyToLastExitRegister:=FALSE,
						bRotateEntranceRegisterBefore:=FALSE,
						bNoKeepTryingMove:=TRUE,
						bTriggerCap:=FALSE,
						bReset:=bResetStates,
						iEntranceArrayElements:=2,
						iExitArrayElements:=8,
						bInvertWriting:=FALSE,
						eClearPackageState:=eClearPackageState,
						bTriggerCounter:=bMRCapCorrect,
						eEntranceState:=eAfterScrewerPackageState,
						//eExitState:=eUnderCorrectCapPackageState, //dd do testów USUNAĆ
						eExitState:=eUnderCorrectCapPackageStateTemp,						
						bKeepTryingMove:=bKeepTryingMove1,
						bError=>,
						iError=>,
						bTriggerDone=>,
						bTriggerFilteredOUT=>);			

eUnderCorrectCapPackageStateTemp[1]:= eClearPackageState; //dd do testów USUNAĆ
eUnderCorrectCapPackageStateTemp[2]:= eClearPackageState;//dd do testów USUNAĆ 
						
// (4) Przesuwanie formatek spod zakrecearek za zakrecarki  
//rtfbFormsDragingPneumaticStationDragging(CLK:=P10_GripperScrewer.fbGripperScrewersDragStation.eRunningState = E_DragStationState.eDraging);
rtfbFormsDragingPneumaticStationDragging(CLK:=P10_GripperScrewer.fbGripperScrewersDragStation.eRunningState = E_DragStationState.eDraging AND P10_GripperScrewer.fbGripperScrewersDragStation.lrActualDragPosition>80);

IF rtfbFormsDragingPneumaticStationDragging.Q THEN
	eAfterScrewerPackageState[1]		:=	eUnderScrewerPackageState[1];
	eAfterScrewerPackageState[2]		:=	eUnderScrewerPackageState[2];
	eUnderScrewerPackageState[1]		:=	eClearPackageState;
	eUnderScrewerPackageState[2]		:=	eClearPackageState;
END_IF

								
// (5) Przesuwanie formatek sprzed zakrecarek na zakrecarki
IF rtfbFormsDragingPneumaticStationDragging.Q THEN
	eUnderScrewerPackageState[1]		:=	eBeforeScrewersPackageState[1];
	eBeforeScrewersPackageState[1]		:=	eClearPackageState;
	eUnderScrewerPackageState[2]		:=	eBeforeScrewers2PackageState[1];
	eBeforeScrewers2PackageState[1]		:=	eClearPackageState;
END_IF

// (6) Przesuwanie formatek zza sprawdzania zalozenia na przed zakrecarki
fbIbScrewerThirdFormCheckFormSensor			(bIN:= 	P10_GripperScrewer.IbGripperScrewersThirdFormCheckFormSensor,		tFilterTimeOn:=T#30MS,	tFilterTimeOff:=T#30MS); //BYŁO 20ms
ftfbIbScrewerThirdFormCheckFormSensor		(CLK:=	fbIbScrewerThirdFormCheckFormSensor.bOUT, 			Q=>);
rtfbIbScrewerThirdFormCheckFormSensor		(CLK:=	fbIbScrewerThirdFormCheckFormSensor.bOUT, 			Q=>);
bTrendIbThirdFormCheckFormSensor:=P10_GripperScrewer.IbGripperScrewersThirdFormCheckFormSensor;
bTrendFilteredIbThirdFormCheckFormSensor:=ftfbIbScrewerThirdFormCheckFormSensor.Q;
ftbMRBeforeScrewer2Block 					(CLK:=	bMRBeforeScrewer2Block,								Q=>);
tofftbMRBeforeScrewer2Block					(IN:=	ftbMRBeforeScrewer2Block.Q,							PT:=T#1100MS);//bylo 350		//  bylo 1000			


// Ustawianie blokady dla ruchu tylko w jedną stronę siłownika
IF ( P10_GripperScrewer.fbGripperScrewersDragStation.eRunningState = E_DragStationState.eDraging )
	AND NOT bMRBeforeScrewer2Block AND NOT tofftbMRBeforeScrewer2Block.Q THEN
	bMRBeforeScrewer2Block := TRUE;
END_IF

//IF bMRBeforeScrewer2Block AND P00_PackML.tonGripperScrewerDragMiddleSensor.Q THEN
IF bMRBeforeScrewer2Block AND P10_GripperScrewer.fbGripperScrewersDragStation.eRunningState = E_DragStationState.eDraging AND P10_GripperScrewer.fbGripperScrewersDragStation.lrActualDragPosition>90 THEN	
	bMRBeforeScrewer2Block := FALSE;
END_IF


//(6)
fbMRBeforeScrewer2PackageState(
                        bFirstCycle:= GVL.bFirstCycle,
                        bTrigger:=ftfbIbScrewerThirdFormCheckFormSensor.Q AND NOT bMRBeforeScrewer2Block,
                        tTriggerFilterTimeOn:=T#0MS,
                        tTriggerFilterTimeOff:=T#0MS,
                        bTriggerBottle:=FALSE,
                        bWithBottleControl:=FALSE,
                        bWithCapControl:=FALSE,
                        bWithFormControlTrigerCounter:=FALSE,
                        bRotateEntranceRegisterBefore:=FALSE,
                        bNoKeepTryingMove:=TRUE,
                        bTriggerCap:=,
                        bReset:=bResetStates,
                        iEntranceArrayElements:=2,
                        iExitArrayElements:=2,
                        bInvertWriting:=FALSE,
                        eClearPackageState:=eClearPackageState,
                        bTriggerCounter:=bMRFormInCap,
                        eEntranceState:=eBeforeScrewers2PackageState,
                        eExitState:=eBeforeScrewersPackageState,
                        bKeepTryingMove:=bKeepTryingMove2,
                        bError=>,
                        iError=>,
                        bTriggerDone=>,
                        bTriggerFilteredOUT=>);   										

// (6) A - Dodatkowe przesuniecie na zboczne narastajace
IF rtfbIbScrewerThirdFormCheckFormSensor.Q AND NOT eBeforeScrewers2PackageState[1].bFormPresent THEN
	eBeforeScrewers2PackageState[1] := eBeforeScrewers2PackageState[2];
	eBeforeScrewers2PackageState[2] := eClearPackageState;
END_IF

						
//(7) Przesuwanie formatek spod sprawdzania zalozenia na przed zakrecarki
fbIbCapPuttedCheckFormSensor		(bIN:= 	P09_CapPuttedCheck.IbCapPuttedCheckFormSensor,		tFilterTimeOn:=T#30MS,	tFilterTimeOff:=T#30MS); //Było 20ms
fbIbCapPuttedCheckFormSensorv2		(bIN:= 	P09_CapPuttedCheck.IbCapPuttedCheckFormSensor,		tFilterTimeOn:=T#30MS,	tFilterTimeOff:=T#30MS); //Było 20ms
ftfbIbCapPuttedCheckFormSensor		(CLK:=	fbIbCapPuttedCheckFormSensorv2.bOUT, 					Q=>);

IF ftfbIbCapPuttedCheckFormSensor.Q THEN
	iftfbIbCapPuttedCheckFormSensor := iftfbIbCapPuttedCheckFormSensor+1;
END_IF


bBitTestOn:=TRUE;


fbMRBeforeScrewerPackageState(
                        bFirstCycle:= GVL.bFirstCycle,
                        bTrigger:= ftfbIbCapPuttedCheckFormSensor.Q,
                        tTriggerFilterTimeOn:=T#0MS,
                        tTriggerFilterTimeOff:=T#0MS,
                        bWithCapControl:=TRUE,
                      	bNoKeepTryingMove:=TRUE,
                        bTriggerCap:=P09_CapPuttedCheck.eCapPuttedCheckRunningState = E_CheckerState.eCapOK,
                        bReset:=bResetStates,
                        iEntranceArrayElements:=1,
                        iExitArrayElements:=2,
                        eClearPackageState:=eClearPackageState,
                        eEntranceState:=eBeforeCapControlPackageState,
                        eExitState:=eBeforeScrewers2PackageState,
                        bKeepTryingMove:=bKeepTryingMove3,
						bRFIDReaded:=bRFIDSBeforeScrewerWriteToRegister(*bBitTestOn*), // Ustawiany jeżeli Dane z tablicy RFID zostały wpisane do zwykłego rejestru
                        iBottleWithoutCap:=iCapFeederCheckCountNOK,
						bError=>,
                        iError=>,
                        bTriggerDone=>,
                        bTriggerFilteredOUT=>);   
				


// --------------------------------------

aCycleRegisterROPP();

// (7,5-7,8) Przesuwanie pod sorterem nasadek

aCycleRegisterCapSorter();

// --------------------------------------

